(* CODESYS project КАРКАС_СПК_107_М01_07_SP_14_temp-3.project

Project tree, tasks and I/O mapping:
  Device : SPK1xx[M01], Production association OWEN, order no. 4, version 3.5.14.34
    application Application
      libraries: Standard, * (System); ComService, 3.5.4.2 (OWEN); SysCom, 3.5.5.0 (System); ModBus, 3.5.4.3 (Production association OWEN); VisuDialogs, * (System); SysFile, 3.5.9.0 (System); Util, * (System); BASIC, 3.3.3.0 (OSCAT); Visu Utils, 3.5.12.0 (System); AlarmManager, 3.5.14.0 (Intern)
      task VISU_TASK (cyclic, interval 100 ms, priority 30) calls VisuElems.Visu_Prg
      task AlarmManagerTask (cyclic, interval 50 ms, priority 1) calls AlarmManager.Alarm_Prg
      task COM3_TASK (freewheeling, priority 4) calls COM3_PRG
      task MainTask (cyclic, interval t#20ms, priority 5) calls CURRENT_PRG [Обработка непрерывных функций], ASDA_PRG [Обработка алгоритмы работы сервопривода головки]
      task COM2_TASK (freewheeling, priority 3) calls COM2_PRG
      task COM1_TASK (freewheeling, priority 2) calls COM1_PRG [Чтение и запись регистров ASDA-A2 и DVP-SS2]
      program COM3_PRG [ST]
      text list AsdaTextList
      global variables GVL
      STRUCT/
        data type TChiller
        data type TWriteCmd
        data type TSetts
        data type TPulling
        data type TReg
        data type DInt_Word
        data type TModbusRegs
        data type TRWRegs
        data type TAsdaParams
        data type TShnek
        data type TAsda
        data type TReadCmd
        data type TDvp
        data type TPeriod
        data type TPID
        data type TNagrev
        data type TTable
        data type TProject
      SRC_AUX/
        function SWAP_BYTES [ST]
        function BYTES_FROM_DINT [ST]
        function HiWord [ST]
        function LoWord [ST]
        function LoByte [ST]
        function HiByte [ST]
        function BYTES_FROM_INT [ST]
      text list DvpTextList
      SRC_FILE/
        function WRITE_OPTIONS [ST]
        function READ_OPTIONS [ST]
        function RECORD_SAVE [ST]
        function RECS_SELECT [ST]
        function REC_DELETE [ST]
        function REC_EXCHANGE [ST]
        function REC_NAME_EXISTS [ST]
      image pool ImagePool
      SRC/
        program AddReadCmd [ST]
        function SET_FRAME_INDEX_EX [CFC]
        function IsRegValid [ST]
        function ButtonColor [ST]
        program AsdaSetParams [ST]
        function BYTES_FROM_WORD [ST]
        function MERGE_RGB [ST]
        function SET_FRAME_INDEX [CFC]
        program ProcessTempers [ST]
        function WORD_FROM_BYTES [ST]
        function INT_FROM_BYTES [ST]
        function QueuePopReg [ST]
        function QueuePushReg [ST]
        function GET_SET_TEMPERS [ST]
        function block AddWriteCmd_FB [ST]
        function KEYBOARD_STR [ST]
        program ASDA_INIT [ST]
        program ASDA_PARAMS [ST]
        program ASDA_HOMING [ST]
        program ASDA_PULSING [ST]
        program ASDA_SERVO_ON [ST]
        program ASDA_SERVO_OFF [ST]
        program ASDA_PARKING [ST]
        function TERNAR_INT [ST]
        program ASDA_STOP [ST]
        function PENTAR_INT [ST]
        function block PROCESS_DELAY_FB [ST]
      Visu/
        visualisation VIS_SETTS_2
        visualisation Main_Panel
        visualisation DlgConfirm
        visualisation Panel_Reg
        visualisation VIS_MSGS
        visualisation VIS_SETTS_4
        visualisation Setts_Panel
        visualisation VIS_REG
        visualisation VIS_PERIOD
        visualisation VIS_OPERATOR
        visualisation DlgPids
        visualisation VIS_SETTS_1
        visualisation VIS_SETTS_3
        visualisation DlgPulling
        visualisation DlgTargetRegParams
        visualisation DlgConfirmAsdaCMD
        visualisation DlgRegLoad
        visualisation DlgShow
        visualisation DlgKeyboard
        visualisation DlgConfirmSaveAS
        visualisation VIS_EDITOR
        visualisation DlgDeleteRec
      program COM1_PRG [ST]
      global variables GVL_FILE
      program COM2_PRG [ST]
      Alarm Configuration
        alarm class ERR_PCHV (priority 10, acknowledge REP)
        alarm class ERR_PVOZD (priority 10, acknowledge REP)
        text list AG_DVP
        alarm class WARN (priority 10, acknowledge REP)
        alarm group AG_DVP
            1 [ERR_DVP]: Comparison Equal, ExpressionToCompare TRUE, Expression Dvp.E_BITS_si.1 - "Зажим не на исходном концевике"
            2 [ERR_DVP]: Comparison Equal, ExpressionToCompare TRUE, Expression Dvp.E_BITS_si.2 - "Нож не на исходном концевике"
            3 [ERR_DVP]: Comparison Equal, ExpressionToCompare TRUE, Expression Dvp.E_BITS_si.3 - "Превышено время движения зажима"
            4 [ERR_DVP]: Comparison Equal, ExpressionToCompare TRUE, Expression Dvp.E_BITS_si.4 - "Превышено время схода ножа с исходного концевика"
            5 [ERR_DVP]: Comparison Equal, ExpressionToCompare TRUE, Expression Dvp.E_BITS_si.5 - "Превышено время возврата каретки на исходный концевик"
            11 [WARN]: Comparison Equal, ExpressionToCompare FALSE, Expression Dvp.STOP_MANUAL_si - "Нажата аварийная кнопка !"
            7 [ERR_DVP]: Comparison Equal, ExpressionToCompare TRUE, Expression Dvp.E_BITS_si.7 - "РЕЗЕРВ"
            6 [ERR_DVP]: Comparison Equal, ExpressionToCompare TRUE, Expression Dvp.E_BITS_si.6 - "Каретка в крайнем положении"
            8 [WARN]: Comparison Equal, ExpressionToCompare TRUE, Expression Dvp.E_BITS_si.8 - "Превышено время схода каретки с исходного концевика"
            9 [WARN]: Comparison Equal, ExpressionToCompare TRUE, Expression Dvp.E_BITS_si.9 - "Превышено время движения ножа"
            10 [WARN]: Comparison Equal, ExpressionToCompare TRUE, Expression ALARM_MOVE - "Нет движения заготовки в тянущем устройстве"
            0 [ERR_DVP]: Comparison Equal, ExpressionToCompare TRUE, Expression Dvp.E_BITS_si.0 - "Каретка не на исходном концевике"
        text list AG_CONNECT
        alarm group AG_AVAR
            0 [ERR_TEMP]: Comparison Equal, ExpressionToCompare TRUE, Expression Nagrev.E_critical_high - "Превышена критическая температура одной из зон"
            1 [ERR_TEMP]: Comparison Equal, ExpressionToCompare TRUE, Expression Nagrev.E_critical_low - "Температура одной из зон ниже температуры запуска привода"
            2 [WARN]: Comparison Equal, ExpressionToCompare TRUE, Expression Nagrev.E_temp_high - "Превышена температура одной из зон"
            3 [WARN]: Comparison Equal, ExpressionToCompare TRUE, Expression Nagrev.E_temp_low - "Низкая температура одной из зон"
        text list MSGS
        alarm class ERR_CHILLER (priority 10, acknowledge REP)
        alarm class ERR_TEMP (priority 10, acknowledge REP)
        alarm class ERR_DVP (priority 10, acknowledge REP)
        alarm group AG_DEV
            0 [ERR_ASDA]: Comparison Equal, ExpressionToCompare TRUE, Expression Asda.E_CODE.0 - "Сигнал аварии от сервопривода"
            1 [ERR_ASDA]: Comparison Equal, ExpressionToCompare TRUE, Expression Asda.E_CODE.1 - "Сигнал предупреждения от сервопривода"
            2 [ERR_ASDA]: Comparison Equal, ExpressionToCompare TRUE, Expression Asda.E_CODE.2 - "Ошибка инициализации Р2-30 или Р3-06"
            3 [ERR_ASDA]: Comparison Equal, ExpressionToCompare TRUE, Expression Asda.E_CODE.3 - "Превышено время операции HOMING"
            4 [ERR_ASDA]: Comparison Equal, ExpressionToCompare TRUE, Expression Asda.E_CODE.4 - "Превышено время операции ПАРКОВКА"
            5 [WARN]: Comparison Equal, ExpressionToCompare TRUE, Expression Asda.E_CODE.5 - "Ограничение момента сервопривода головки"
            6 [MSG]: Comparison Equal, ExpressionToCompare TRUE, Expression Asda.E_CODE.6 - "Тестовая ошибка"
            7 [ERR_PCHV]: Comparison Equal, ExpressionToCompare TRUE, Expression ALARM_PCHVS.0 - "Аварийный сигнал ПЧВ шнека"
            10 [ERR_PCHV]: Comparison Equal, ExpressionToCompare TRUE, Expression ALARM_PCHVS.8 - "Аварийный сигнал ПЧВ тянущего устройства"
        alarm class MSG (priority 10, acknowledge REP)
        alarm class ERR_ASDA (priority 10, acknowledge REP)
        alarm group AG_CONNECT
            0 [ERR_CONNECT]: Comparison Equal, ExpressionToCompare FALSE, Expression Asda.Connect - "Нет соединение с сервоприводом ASDA-A2"
            1 [ERR_CONNECT]: Comparison Equal, ExpressionToCompare FALSE, Expression Dvp.Connect - "Нет соединения с контроллером DVP"
            2 [ERR_CONNECT]: Comparison Equal, ExpressionToCompare FALSE, Expression Shnek.Connect - "Нет соединения с ПЧВ шнека"
            3 [ERR_CONNECT]: Comparison Equal, ExpressionToCompare FALSE, Expression Pulling.Connect - "Нет соединения с ПЧВ тянущего устройства"
            4 [ERR_CONNECT]: Comparison Equal, ExpressionToCompare FALSE, Expression Chiller.Connect - "Нет соединения с Чиллером"
        text list AG_AVAR
        alarm class ERR_CONNECT (priority 10, acknowledge REP)
        alarm group AG_MSGS
            1 [MSG]: Comparison Equal, ExpressionToCompare TRUE, Expression Dvp.bunker_viveden_msg
            3 [MSG]: Comparison Equal, ExpressionToCompare FALSE, Expression Dvp.Uroven_s_si
            4 [ERR_PVOZD]: Comparison Equal, ExpressionToCompare FALSE, Expression Dvp.PVozd_si
            5 [MSG_PCHV]: Comparison Equal, ExpressionToCompare TRUE, Expression ALARM_PCHVS.1
            11 [MSG_PCHV]: Comparison Equal, ExpressionToCompare TRUE, Expression ALARM_PCHVS.11
            7 [MSG_PCHV]: Comparison Equal, ExpressionToCompare TRUE, Expression ALARM_PCHVS.3
            6 [MSG_PCHV]: Comparison Equal, ExpressionToCompare TRUE, Expression ALARM_PCHVS.2
            12 [MSG_PCHV]: Comparison Equal, ExpressionToCompare TRUE, Expression ALARM_PCHVS.12
            13 [MSG]: Comparison Equal, ExpressionToCompare FALSE, Expression Dvp.Uroven_w_si
            8 [MSG_PCHV]: Comparison Equal, ExpressionToCompare TRUE, Expression ALARM_PCHVS.4
            9 [MSG_PCHV]: Comparison Equal, ExpressionToCompare TRUE, Expression ALARM_PCHVS.9
            10 [MSG_PCHV]: Comparison Equal, ExpressionToCompare TRUE, Expression ALARM_PCHVS.10
            0 [MSG]: Comparison Equal, ExpressionToCompare TRUE, Expression Nagrev.Temper_reached_msg
        text list AG_DEV
        text list AG_CHILLER
        alarm group AG_CHILLER
            11 [ERR_CHILLER]: Comparison Equal, ExpressionToCompare TRUE, Expression Chiller.AlarmFlag1.11 - "Низкая температура нагревания Чиллера"
            21 [ERR_CHILLER]: Comparison Equal, ExpressionToCompare TRUE, Expression Chiller.AlarmFlag2.5 - "Неисправность датчика температуры на выходе Чиллера"
            31 [ERR_CHILLER]: Comparison Equal, ExpressionToCompare TRUE, Expression Chiller.AlarmFlag2.15 - "Обнаружен сигнал контакта входа 2 Чиллера"
            14 [ERR_CHILLER]: Comparison Equal, ExpressionToCompare TRUE, Expression Chiller.AlarmFlag1.14 - "Падение давления на высокой стороне контура хладагента Чиллера"
            24 [ERR_CHILLER]: Comparison Equal, ExpressionToCompare TRUE, Expression Chiller.AlarmFlag2.8 - "Неисправность датчика давления нагнетания Чиллера"
            34 [ERR_CHILLER]: Comparison Equal, ExpressionToCompare TRUE, Expression Chiller.AlarmFlag3.2 - "Неисправен датчик элетрического сопротивления жидкости в Чиллере"
            19 [ERR_CHILLER]: Comparison Equal, ExpressionToCompare TRUE, Expression Chiller.AlarmFlag2.3 - "Ошибка памяти контроллера Чиллера"
            29 [ERR_CHILLER]: Comparison Equal, ExpressionToCompare TRUE, Expression Chiller.AlarmFlag2.13 - "Обслуживание компрессора двигателя Чиллера"
            17 [ERR_CHILLER]: Comparison Equal, ExpressionToCompare TRUE, Expression Chiller.AlarmFlag2.1 - "Перегрузка компрессора Чиллера"
            27 [ERR_CHILLER]: Comparison Equal, ExpressionToCompare TRUE, Expression Chiller.AlarmFlag2.11 - "Обслуживание насоса Чиллера"
            12 [ERR_CHILLER]: Comparison Equal, ExpressionToCompare TRUE, Expression Chiller.AlarmFlag1.12 - "Высокое давление нагнетания компрессора Чиллера"
            22 [ERR_CHILLER]: Comparison Equal, ExpressionToCompare TRUE, Expression Chiller.AlarmFlag2.6 - "Неисправность датчика температуры на входе Чиллера"
            32 [ERR_CHILLER]: Comparison Equal, ExpressionToCompare TRUE, Expression Chiller.AlarmFlag3.0 - "Обнаружена утечка воды Чиллера"
            15 [ERR_CHILLER]: Comparison Equal, ExpressionToCompare TRUE, Expression Chiller.AlarmFlag1.15 - "Повышение давления на низкой стороне контура хладагента Чиллера"
            25 [ERR_CHILLER]: Comparison Equal, ExpressionToCompare TRUE, Expression Chiller.AlarmFlag2.9 - "Неисправность датчика давления нагнетания компрессора Чиллера"
            16 [ERR_CHILLER]: Comparison Equal, ExpressionToCompare TRUE, Expression Chiller.AlarmFlag2.0 - "Падение давления на низкой стороне контура хладагента Чиллера"
            10 [ERR_CHILLER]: Comparison Equal, ExpressionToCompare TRUE, Expression Chiller.AlarmFlag1.10 - "Низкая температура на входе компрессора Чиллера"
            20 [ERR_CHILLER]: Comparison Equal, ExpressionToCompare TRUE, Expression Chiller.AlarmFlag2.4 - "Сработал предохранитель постоянного тока в Чиллере"
            30 [ERR_CHILLER]: Comparison Equal, ExpressionToCompare TRUE, Expression Chiller.AlarmFlag2.14 - "Обнаружен сигнал контакта входа 1 Чиллера"
            13 [ERR_CHILLER]: Comparison Equal, ExpressionToCompare TRUE, Expression Chiller.AlarmFlag1.13 - "Unused"
            23 [ERR_CHILLER]: Comparison Equal, ExpressionToCompare TRUE, Expression Chiller.AlarmFlag2.7 - "Неисправность датчика температуры на входе компрессора Чиллера"
            33 [ERR_CHILLER]: Comparison Equal, ExpressionToCompare TRUE, Expression Chiller.AlarmFlag3.1 - "Повышение элетрического удельного сопротивления жидкости в Чиллере"
            18 [ERR_CHILLER]: Comparison Equal, ExpressionToCompare TRUE, Expression Chiller.AlarmFlag2.2 - "Ошибка связи с контроллером Чиллера"
            28 [ERR_CHILLER]: Comparison Equal, ExpressionToCompare TRUE, Expression Chiller.AlarmFlag2.12 - "Обслуживание вентилятора двигателя Чиллера"
            8 [ERR_CHILLER]: Comparison Equal, ExpressionToCompare TRUE, Expression Chiller.AlarmFlag1.8 - "Падение давления нагнетания Чиллера"
            9 [ERR_CHILLER]: Comparison Equal, ExpressionToCompare TRUE, Expression Chiller.AlarmFlag1.9 - "Высокая температура на входе компрессора Чиллера"
            26 [ERR_CHILLER]: Comparison Equal, ExpressionToCompare TRUE, Expression Chiller.AlarmFlag2.10 - "Неисправность датчика давления на входе компрессора Чиллера"
            0 [ERR_CHILLER]: Comparison Equal, ExpressionToCompare TRUE, Expression Chiller.AlarmFlag1.0 - "Низкий уровень воды в Чиллере"
            1 [ERR_CHILLER]: Comparison Equal, ExpressionToCompare TRUE, Expression Chiller.AlarmFlag1.1 - "Высокая температура воды на выходе Чиллера"
            2 [ERR_CHILLER]: Comparison Equal, ExpressionToCompare TRUE, Expression Chiller.AlarmFlag1.2 - "Температура на выходе Чиллера выросла"
            3 [ERR_CHILLER]: Comparison Equal, ExpressionToCompare TRUE, Expression Chiller.AlarmFlag1.3 - "Температура на выходе Чиллера..."
            4 [ERR_CHILLER]: Comparison Equal, ExpressionToCompare TRUE, Expression Chiller.AlarmFlag1.4 - "Высокая температура воды на входе Чиллера"
            5 [ERR_CHILLER]: Comparison Equal, ExpressionToCompare TRUE, Expression Chiller.AlarmFlag1.5 - "Высокая давление нагнетания Чиллера"
            6 [ERR_CHILLER]: Comparison Equal, ExpressionToCompare TRUE, Expression Chiller.AlarmFlag1.6 - "Ненормальная работа насоса Чиллера"
            7 [ERR_CHILLER]: Comparison Equal, ExpressionToCompare TRUE, Expression Chiller.AlarmFlag1.7 - "Повышение давления нагнетания Чиллера"
        alarm class MSG_PCHV (priority 10, acknowledge REP)
        text list AlarmGroup
        alarm group AlarmGroup
      program CURRENT_PRG [ST]
      text list FileTextList
      program ASDA_PRG [ST]
    Network : Network, Production association OWEN, version 3.5.14.3001
        unmapped channels: DHCP enabled, IP, Mask, Gateway, MAC, Hostname, Enable DHCP, New IP, New Mask, New Gateway, New Hostname, Set Settings
    Drives : Drives, Production association OWEN, version 3.5.14.3001
        input  Application.MMCMounted : BIT  // MMC Mounted
        output Application.EnableDrivers : BIT  // Enable Drives
        output Application.bUnmount : BIT  // MMC Unmount
        unmapped channels: FS size, FS used, FS free, USB Mounted, USB Unmount done, USB size, USB used, USB free, MMC Unmount done, MMC size, MMC used, MMC free, USB Unmount
    Buzzer : Buzzer, Production association OWEN, version 3.5.14.3001
        unmapped channels: Buzzer enabled, Enable Buzzer
    Info : Info, Production association OWEN, version 3.5.14.3001
        input  Application.Project.sVendor : ARRAY [0..80] OF BYTE  // VENDOR
        input  Application.Project.sName : ARRAY [0..80] OF BYTE  // DEVICE
        input  Application.Project.sSerial : ARRAY [0..80] OF BYTE  // SERIAL
        input  Application.Project.sRuntime : ARRAY [0..80] OF BYTE  // RUNTIME
        input  Application.Project.sFirmwareVersion : ARRAY [0..80] OF BYTE  // FIRMWARE
        input  Application.Project.sLinuxVersion : ARRAY [0..80] OF BYTE  // LINUX
        input  Application.Project.sNeedTarget : ARRAY [0..80] OF BYTE  // TARGET
        unmapped channels: PROJECT, AUTHOR, VERSION, PROFILE, LASTCHANGES
    Debug : Debug, Production association OWEN, version 3.5.14.3001
        unmapped channels: RAM used, RAM free, Open files, Processor usage, Core temp, Enable Debug, Debug pause
    OwenCloud : OwenCloud, Production association OWEN, version 3.5.14.3002
        unmapped channels: OwenCloud enabled, Folder error, Symbol error, No Symbol Config, Status, Enable OwenCloud
    Screen : Screen, Production association OWEN, version 3.5.14.3001
        unmapped channels: Get Brightness, Dim time, Off time, Full brightness, Dim brightness, Off brightness, Dim visu name, Off visu name, On visu name, Wake up
    OwenRTC : OwenRTC, Production association OWEN, version 3.5.14.3001
        unmapped channels: Year, Month, Day, Hour, Minute, Second, Day of Week, Week of Year, Format Date, Format Time, UTC Offset, NTP Enabled, NTP Error, System Timer, Date And Time, New Year, New Month, New Day, New Hour, New Minute, New Second, New UTC Offset, Set Settings DT, Enable NTP, Prefer Server
    Watchdog : Watchdog, Production association OWEN, version 3.5.14.3001
        unmapped channels: Exception Handling, Last Exception Code, Last Exception Description, Last Exception Time, Hardware Watchdog Flag, Power Reboot Count, Watchdog Reboot Count, Exception Reboot Count, Command Reboot Count, Reboot, Reset Counters
  5ce3da45-db07-42e7-a21c-a00fff4ed8f6|Images\Banned.png
  5ce3da45-db07-42e7-a21c-a00fff4ed8f6|Images\crosscirclehd.png
  5ce3da45-db07-42e7-a21c-a00fff4ed8f6|Images\Good.png
  5ce3da45-db07-42e7-a21c-a00fff4ed8f6|Images\Dialog_win_7_800x480.jpg
  5ce3da45-db07-42e7-a21c-a00fff4ed8f6|Images\Dialog_win_7_400x200.jpg
  5ce3da45-db07-42e7-a21c-a00fff4ed8f6|Images\iError.png
  5ce3da45-db07-42e7-a21c-a00fff4ed8f6|Images\tickcirclehd.png
  5ce3da45-db07-42e7-a21c-a00fff4ed8f6|Images\danger.png
  5ce3da45-db07-42e7-a21c-a00fff4ed8f6|Images\Dialog_win_7_600x300.jpg
  text list GlobalTextList
  5ce3da45-db07-42e7-a21c-a00fff4ed8f6|Images\Warning.png
  5ce3da45-db07-42e7-a21c-a00fff4ed8f6|Images\Dialog_win_7_700x380.jpg
  5ce3da45-db07-42e7-a21c-a00fff4ed8f6|Images\Dialog_win_7_750x450.jpg
*)

// Device/Application/STRUCT/TChiller
TYPE TChiller :
STRUCT
	Connect			: BOOL;			// Флаг соединения с Чиллером
	T_ACTUAL		: REAL;
	
	Pusk			: BOOL;
	Block			: BOOL;
	AVAR			: BOOL;			// Флаг аварии Чиллера (читаем по RS-485)
	Status			: WORD;
	Status_2		: WORD;

	AlarmFlag1		: WORD;			// Флаги аварии Чиллера
	AlarmFlag2		: WORD;
	AlarmFlag3		: WORD;

	FillColor		: DWORD;		(* Цвет заливки окошка температуры *)
	FrameColor		: DWORD;		(* Цвет контура окошка температуры *)

	BtnFillColor	: DWORD;		(* Цвет заливки площадок кнопок ПУСК в автоматическом режиме *)
	BtnFrameColor	: DWORD;		(* Цвет контура площадок кнопок ПУСК в автоматическом режиме *)
	
END_STRUCT
END_TYPE

(*
Status flag

0	Run flag						Run status (Include the independent operation of the pump) 0= Stop 1= Run
1	Operation stop alarm flag		Operation stop alarm given off status 0= Not occurred 1= Operation stop alarm given off
2 	Operation continued alarm flag	Operation continued alarm given off status 0= Not occurred 1= Operation continued alarm given off
3	Unused
4	Press Unit flag					Pressure unit set status 0= MPa 1= PSI
5	Remote status flag				Remote status 0= Other than SERIAL mode 1= SERIAL mode
6	Unused
7	Unused
8	Unused
9	Completion of preparation		Completion of preparation (TEMP READY) status
	(TEMP READY) flag				0= Condition isn’t formed 1= Condition is formed
10	Temperature unit flag			Temperature unit set status 0= Centigrade (oC) 1= Fahrenheit (oF)
11	Run timer flag					Run timer set status 0= Not set 1= Set
12	Stop timer flag					Stop timer set status 0= Not set 1= Set
13	Reset after power failure flag	Reset after power failure set status 0= Not set 1= Set
14	Anti-freezing flag				Anti-freezing set status 0= Not set 1= Set
15	Automatic fluid filling flag	Automatic fluid filling condition 0= Stop 1= Fluid ∗ The signal of the product without an option [Automatic filling] also changes.

Status flag 2
0-1	Electric resistivity/			Electric resistivity/conductivity setting status conductivity setting flag
									0= Not set 1= Electric resistivity is set 2= Electric conductivity is set
2-15	Unused
*)

// Device/Application/STRUCT/TWriteCmd
TYPE TWriteCmd :
(
	wcAsda_P2_30:=0,
	wcAsda_P3_06,
	wcAsda_P4_07_1,
	wcAsda_P4_07_2,
	wcAsda_P4_07_3,
	wcAsda_P4_07_4,
	
	wcAsdaParams,
	wcAsda_Homing,
	wcAsda_Forward,
	wcAsda_Backward,
	wcAsda_Parking,
	wcAsda_Working,
	wcAsda_Stop,
	
	wcChiller_Ust,
	wcChiller_Start,
	wcChiller_Stop,
	
	wcShnek_Ust,
	wcShnek_Start,
	wcShnek_Stop,
	
	wcPulling_Ust,
	wcPulling_Start,
	wcPulling_Stop
);
END_TYPE

// Device/Application/STRUCT/TSetts
TYPE TSetts :
STRUCT
	T_ZAP					: ARRAY [0..NUM_TEMPS-1] OF REAL;		// Температуры запуска приводов
	TM_VIGON				: WORD;		// Время выгона массы в секундах	
	otkl_alarm_zvuk			: BOOL;		// Флаг отключения звуковой сигнализации аварий
	otkl_h_temp				: BOOL;		// Переменная для отключения ошибки "Превышение температуры одной из зон"
	otkl_l_temp				: BOOL; 	// Переменная для отключения ошибки "Низкая температура одной из зон" 
	otkl_c_pulling			: BOOL;		// Переменная для отключения контроля движения ТЯУ
	use_vigon				: BOOL;		// Флаг выгона массы
	use_bunker				: BOOL;		// Флаг использования бункера
	use_servo_without_temp	: BOOL;		// Разрешить работу головки без разогрева (ТОЛЬКО ДЛЯ ОТЛАДКИ !!!)
	use_shnek_without_temp	: BOOL;		// Разрешить работу шнека без разогрева (ТОЛЬКО ДЛЯ ОТЛАДКИ !!!)
	
	CondEnableZones1_4		: BOOL;		// Флаг для условного включения зон 1-4
	CondIZone				: BYTE;		// Номер зоны (5-7), по которой управляется включение зон 1-4
	CondValue				: REAL;		// Значение 0-100 % от температуры уставки зоны (5-7), при превышении которой включаются зоны 1-4

	REP_MM					: REAL;		// Начальное положение (смещение) реперной точки относительно заднего концевика в 0.01 мм
	TimeVigon				: WORD;		// Время выгона массы после вывода бункера в секундах
	K_Length				: REAL;		// Длина заготовки в мм
	zd_temps				: ARRAY [0..NUM_TEMPS-1] OF REAL;	// Температуры для автонастройки ПИД-регуляторов

END_STRUCT
END_TYPE

// Device/Application/STRUCT/TPulling
TYPE TPulling :
STRUCT
	Connect			: BOOL;			(* Флаг соединения *)
	Pusk			: BOOL;			(* Флаг включения *) 
	Block			: BOOL;			(* Блокировка тянущего *)
	STW				: WORD;			(* Слово состояния *)
	MAV				: WORD;			(* Основное текущее значение привода *)
	
	Speed			: REAL;			(* Реальная скорость движения в процентах *)
	ActiveParamSet	: WORD;			(* Активный набор данных в ПЧВ *)
	BtnFillColor	: DWORD;		(* Цвет заливки площадок кнопок ПУСК в автоматическом режиме *)
	BtnFrameColor	: DWORD;		(* Цвет контура площадок кнопок ПУСК в автоматическом режиме *)
	
	
END_STRUCT
END_TYPE

(* ПЧВ ТЯУ использует 2 набора параметров:
Набор параметров 1 - для работы без обратной связи,
Набор параметров 2 - для работы с обратной связью и ПИ-регулятором *)

(*
1. Обороты двигателя ТЯУ при 50 Гц = 1350 об/мин
2. Редуктор - к-т редукции = 304
3. Обороты вала редуктора = 1350/304 = 4,44 об/мин
4. Число зубов ведущей шестерёнки = 11
5. Число зубов ведомой шестерёнки = 20
6. Обороты вала ведомой шестерёнки (тянущего вала) = 4,44*(11/20) = 2,4424 об/мин
7. Диаметр тянущего вала = 97 мм
8. Диаметр шкива энкодера = 63,6 мм
9. Обороты вала энкодера = 2,4424*(97/63,6) = 3,725 об/мин
10. Обороты энкодера в секунду = 3,725,60 = 0,06208 об/сек
11. Частота импульсов энкодера = 0,06208*5000 = 310,425 Гц
12. МАКСИМАЛЬНАЯ ЧАСТОТА ЭНКОДЕРА (при питающей частоте двигателя 100 Гц) = 310,425*100/50 = 620,849 Гц

*)

// Device/Application/STRUCT/TReg
TYPE TReg :
STRUCT
	Name		: STRING (64);						// Имя режима
	Desc		: STRING (64);						// Примечание

	TEMPS		: ARRAY [0..NUM_TEMPS-1] OF REAL;	// Уставки температур зон нагрева 0-6
	T_MASS		: REAL;								// Температура массы
	T_CHIL		: REAL;								// Уставка температуры Чиллера
	Period		: TPeriod;							// Параметры периода работы головки
	
	Qm			: REAL;		// Производительность шнека в процентах (возможно далее в г/мин после экспериментального создания шкалы)
	Speed		: REAL;		// Скорость движения тянущего устройства в процентах (возможно далее в мм / сек)
	Freq		: REAL;		// Частота колебаний коронки, Гц 
	
	REZ_1		: REAL;		// Резерв 1
	REZ_2		: REAL;		// Резерв 2
	REZ_3		: REAL;		// Резерв 3
	
END_STRUCT
END_TYPE

// Device/Application/STRUCT/DInt_Word
TYPE DInt_Word :
UNION

	dDInt	: DINT;
	wWord	: ARRAY[0..1] OF WORD;
	
END_UNION
END_TYPE

// Device/Application/STRUCT/TModbusRegs
TYPE TModbusRegs :
STRUCT
	DevAdr		: BYTE;						// Адрес устройства
	RegAdr		: WORD;						// Адрес регистра
	pVals		: POINTER TO WORD;			// Указатели на переменные (для чтения и записи)
	RegsCount	: BYTE;						// Число регистров записи или чтения
END_STRUCT
END_TYPE

// Device/Application/STRUCT/TRWRegs
TYPE TRWRegs :
STRUCT
	REGS	: ARRAY [0..MAX_MODBUS_REGS-1] OF TModbusRegs;		// Структура для последовательной записи
	Count	: BYTE;												// Счётчик для обработки цикла

END_STRUCT
END_TYPE

// Device/Application/STRUCT/TAsdaParams
//{attribute 'qualified_only'}
//{attribute 'strict'}
TYPE TAsdaParams :
(
	ap_Accs,
	ap_Speeds,
	ap_Dels,
	ap_Dists
);
END_TYPE

// Device/Application/STRUCT/TShnek
TYPE TShnek :
STRUCT
	Connect		: BOOL;			(* Флаг соединения *)
	Pusk		: BOOL;			(* Флаг включения *) 
	Block		: BOOL;			(* Блокировка шнека *)
	STW			: WORD;			(* Слово состояния *)
	MAV			: WORD;			(* Основное текущее значение привода *)
	
	Qm			: REAL;			(* Реальная производительность в процентах *)
	
	FillColor	: DWORD;		(* Цвет заливки площадок кнопок ПУСК в автоматическом режиме *)
	FrameColor	: DWORD;		(* Цвет контура площадок кнопок ПУСК в автоматическом режиме *)

END_STRUCT
END_TYPE

(* Слово состояния STW
---------------------------------------------------------------------
		|		1										|		0
----------------------------------------------------------------------
STW.0	|	Готовность к управлению					|	Управление не готово
STW.1	|	Привод готов							|	Привод не готов
STW.2	|	Нет останова выбегом					|	Останов выбегом
STW.3	|	Аварийный сигнал						|	Нет аварийного сигнала
STW.4	|	Есть отображение ошибки на ЛПО			|	Нет отображения ошибки на ЛПО
STW.5	|	НЕ ИСПОЛЬЗУЕТСЯ							|
STW.6	|	Отключение с блокировкой				|	Нет критических аварий
STW.7	|	Предупреждение							|	Нет предупреждения
STW.8	|	На задании								|	Не на задании (например, разгон)
STW.9	|	Автоматический режим					|	Ручной режим
STW.10	|	В частотном диапазоне					|	Вне частотного диапазона
STW.11	|	Работа									|	Остановлен
STW.12	|	Останов с автоматическим перезапуском	|	Привод в норме
STW.13	|	Предупреждение о напряжении				|	Нет предупреждения о напряжении
STW.14	|	Предел по току							|	Нет предела по току
STW.15	|	Предупреждение о перегреве				|	Нет предупреждения о перегреве

*)

// Device/Application/STRUCT/TAsda
TYPE TAsda :
STRUCT
	Connect			: BOOL;			// Флаг соединения с ASDA-A2
	IsInit			: BOOL;			// Флаг
	IsHoming		: BOOL;			// Флаг нахождения реперной точки
	IsServo_ON		: BOOL;			// Фгаг включенного сервопривода
	DoPulsing		: BOOL;			// Флаг процесса пульсирования
	AllowManual		: BOOL;			// Флаг разрешения ручного режима
	P0_01			: WORD;			// Код ошибки (для логического дополнения до 6 читаемых регистров одной командой через Mapping)
	P0_46			: WORD;			// Параметр P0-46 - состояние дискретных выходов
	P2_30			: WORD;			// Параметр Р2-30 - отключение EEPROM (д.б=5)
	P3_06			: WORD;			// Параметр Р3-06 - способ управления дискретными входами (д.б.=3)
	P4_07			: WORD;			// Параметр Р4-07 - состояние дискретных входов
	P5_07			: WORD;			// Параметр Р5-07 - управление PR - циклическое чтение
	E_CODE			: WORD:=0;		// Код ошибки сервопривода
	WAIT			: BOOL;			// Флаг состояния ожидания
	WAIT_ERR		: BOOL;			// Флаг ожидания команды сброса аварии
	WAIT_WORK		: BOOL;			// Флаг нахождения в состоянии работы
	Pusk			: BOOL;			// Флаг работы в пульсирующем режиме
	Block			: BOOL;			// Блокировка головки
	Torque			: INT;			// Текущий момент
	TorqueMin		: INT;			// Минимальный момент
	TorqueMax		: INT;			// Максимальный момент
	
	// Вспомогательные переменные
	BtnFillColor	: DWORD;	(* Цвет заливки площадок кнопок ПУСК в автоматическом режиме *)
	BtnFrameColor	: DWORD;	(* Цвет контура площадок кнопок ПУСК в автоматическом режиме *)

	text_id			: BYTE;			// Индекс сообщения в списке сообщений - 
	E_ALARM			: WORD;			// Код ошибки сервопривода после перевода из BCD
	
END_STRUCT
END_TYPE

(* Состояние дискретных входов
P4-07.0		- Servo ON
P4-07.1		- Alarm Reset
P4-07.2		- Reverse LIM
P4-07.3		- Forward LIM
*)

(* Коды ошибок сервопривода
E_CODE.0	- SP - сигнал ALRM
E_CODE.1	- SP - сигнал WARN
E_CODE.2	- SP - Ошибка инициализации Р2-30 или Р3-06
E_CODE.3	- SP - Превышено время операции HOMING
E_CODE.4	- SP - Превышено время операции PARKING
E_CODE.5	- SP - Превышение момента
E_CODE.6	- SP - Тестовая ошибка
*)
(* Значения P0-46 (дискретные выходы)
SP_P0_46.0	- SRDY (Готовность привода)
SP_P0_46.1	- SON (Servo On - привод работает)
SP_P0_46.2	- ZSPD (Нулевая скорость)
SP_P0_46.3	- TSPD (Скорость достигнута)
SP_P0_46.4	- TPOS (Зад. положение достигнуто)
SP_P0_46.5	- TQL (Ограничение момента)
SP_P0_46.6	- ALRM (Авария привода)
SP_P0_46.7	- BRKR (Управление тормозом)
SP_P0_46.8	- HOME (Исходное положение достигнуто)
SP_P0_46.9	- OLW (Предупреждение о перегрузке)
SP_P0_46.10	- WARN (Предупреждение активно. WARN активизируется, во время ограничения прямого или обратного вращения;
аварийного стопа, ошибки коммуникации, и при низком напряжении питания.)*)

// Device/Application/STRUCT/TReadCmd
//{attribute 'qualified_only'}
//{attribute 'strict'}
TYPE TReadCmd :
(
	rcAsda_P2_30:=0,		// Дополнительные функции входов		
	rcAsda_P3_06,			// Функция управления входными сигналами
	rcAsda_P6_01			// Положение реперной точки относительно заднего концевика
	
);
END_TYPE

// Device/Application/STRUCT/TDvp
TYPE TDvp :
STRUCT
	Connect				: BOOL;		// Флаг соединения
	bunker_viveden_msg	: BOOL;		// Оповещатель "Бунер выведен !!!"

	Nasos_so			: BOOL;		// Сигнал включения насоса
	Nasos_OTL			: BOOL;		// Флаг отладочного включения насоса

	Uroven_s_si			: BOOL;		// Уровень сырья в бункере
	Uroven_w_si			: BOOL;		// Уровень воды в баке

	Bunker_si			: BOOL;		// Положение бункера
	PVozd_si			: BOOL;		// Давление воздуха
	KarIsx_si			: BOOL;		// Датчик исходного положения каркаса
	KarRab_si			: BOOL;		// Датчик рабочего положения каркаса
	ZazhIsx_si			: BOOL;		// Датчик исходного положения зажима
	KnifeIsx_si			: BOOL;		// Датчик исходного положения ножа
	KnifeRab_si			: BOOL;		// Датчик рабочего положения ножа

	Nasos_si			: BOOL;		// Реле включения насоса
	Karet_si			: BOOL;		// Пневмоцилиндр каретки
	Zazh_si				: BOOL;		// Пневмоцилиндр зажима
	Knife_si			: BOOL;		// Пневмоцидиндр ножа
	F_OTR_si			: BOOL;		// Импульс отрезки заготовки
	STOP_MANUAL_si		: BOOL;		// Сигнал аварийного останова от кнопки СТОП (ИНВЕРСНЫЙ)
	E_BITS_si			: WORD;		// Биты ошибок от DVP

	Pids				: ARRAY [0..NUM_TEMPS-1] OF TPID;		// Параметры ПИД-регуляторов
	pid_index			: WORD;		// Переменная для выбора индекса 0-6 ПИД-регулятора
	zone_index			: WORD;		// Переменная для выбора номера зоны 1-7 ПИД-регулятора
	pid_read			: BOOL;		// Переменная импульса чтения ПИД
	pid_write			: BOOL;		// Переменная импульса записи ПИД
	
	zd_selector			: BOOL;		// Переключатель - откуда брать задания температур для настройки ПИД
	AutoPIDActivate		: BOOL;		// Переменная для активизации автонастройки ПИД
	
	Encoder				: BOOL;		// Флаг вращения энкодера
END_STRUCT
END_TYPE

// Device/Application/STRUCT/TPeriod
TYPE TPeriod :
STRUCT
	Per_FirstHP		: REAL;						// Процент первого полупериода (второй - остаток)
	Per_Pulses		: ARRAY [0..1] OF REAL;		// Проценты импульсов 1-го и 2-го полупериодов в соотв. полупериодах	
	Per_Levels		: ARRAY [0..1] OF REAL;		// Проценты уровней 1-го и 2-го полупериодов в соотв. импульсах
	Offsets			: ARRAY [0..1] OF REAL;		// милиметры, P6-21 - Смещение вперёд, P6-23 - назад от реперной точки
	
END_STRUCT
END_TYPE

(* Единицы измерения
Accs		- милисекунды
Speeds		- обороты в минуту
Dels		- милисекунды
Offsets		- PUU
*)

// Device/Application/STRUCT/TPID
TYPE TPID :
STRUCT
	formula		: WORD;			// Формула ПИД-регулятора (0-независимая, 1-зависимая см. документацию на температурный модуль)
	Kc_Kp		: REAL;			// Пропорциональный коэффициент
	Ti_Ki		: REAL;			// Коэффициент интегрирования
	Td_Kd		: REAL;			// Коэффициент дифференцирования
	Tf			: REAL;			// Постоянная времени дифференцирования
	
END_STRUCT
END_TYPE

// Device/Application/STRUCT/TNagrev
TYPE TNagrev :
STRUCT
	T_Actuals			: ARRAY [0..NUM_TEMPS-1] OF REAL;	// Текущие температуры
	T_ActualMass		: REAL;			// Текущая температура массы
	T_Enables_si		: WORD;			// Биты включенных зон (из Dvp (не используются))
	T_Enables			: WORD;			// Биты заданных включенных зон

	Auto_IN				: BYTE;			// Вспомогательная переменные для сборки сигналов автонастройки от Dvp 
	Auto_OUT			: BYTE;			// Вспомогательная переменная для сборки сигналов автонастройки к Dvp

	E_critical_high		: BOOL;			// Флаг критической температуры одной из зон
	E_critical_low		: BOOL;			// Флаг температуры одной из зон ниже температуры запуска приводов
	E_temp_high			: BOOL;			// Флаг превышения температуры одной из зон
	E_temp_low			: BOOL;			// Флаг низкой температуры одной из зон
	Temper_Reached		: BOOL;			// Флаг выхода на темрературный режим
	Temper_Reached_msg	: BOOL;			// Оповещатель достижения температуры
	Nagrev_on			: BOOL;			// Флаг включения нагревателей
	NagrevFillColor		: DWORD;		// Цвет заливки площадок кнопок ПУСК в автоматическом режиме
	NagrevFrameColor	: DWORD;		// Цвет контура площадок кнопок ПУСК в автоматическом режиме
	FillColors			: ARRAY [0..NUM_TEMPS-1] OF DWORD;	// Массив цветов заливок
	FrameColors			: ARRAY [0..NUM_TEMPS-1] OF DWORD;	// Массив цветов фреймов
	FillColorMass		: DWORD;		// Цвет заливки окошка температуры массы
	FrameColorMass		: DWORD;		// Цвет контура окошка температуры массы

	text_id				: BYTE;			// Индекс текста из списка состояний

END_STRUCT
END_TYPE

// Device/Application/STRUCT/TTable
TYPE TTable :
STRUCT
	Recs		: ARRAY [0..TABLE_NUM_ROWS-1] OF TReg;	// Записи таблицы
	RowCount	: INT;	// Число строк таблицы, RowCount-1 - максимальный индекс массива для таблицы
	RowSel		: INT;	// Выделеная строка в таблице
	PageNum		: INT;	// Номер страницы в таблице 
	NumFileRecs	: INT;	// Суммарное число записей в таблице
	iMsg		: BYTE;	// Флаг сообщений при загрузке таблицы

END_STRUCT
END_TYPE

// Device/Application/STRUCT/TProject
TYPE TProject :
STRUCT
	sVendor				: STRING;	// Производитель
	sName				: STRING;	// Имя
	sSerial				: STRING;	// Серийный номер	
	sRuntime			: STRING;	// Рабочая версия
	sFirmwareVersion	: STRING;	// Информация о прошивке
	sNeedTarget			: STRING;	// Требуемый таргет-файл
	sLinuxVersion		: STRING;	// Версия ОС Linux в контроллере
	
	
	
END_STRUCT
END_TYPE

// Device/Application/GVL
VAR_GLOBAL CONSTANT

ADR_DVP			: BYTE:=1;		// Modbus адрес контроллера DVP на линии COM_1 
ADR_ASDA		: BYTE:=64;		// Modbus адрес сервопривода ASDA на линии COM_1
ADR_SHNEK		: BYTE:=24;		// Modbus адрес  частотника шнека на линии COM_2
ADR_PULLING		: BYTE:=32;		// Modbus адрес  частотника тянущего устройства на линии COM_2
ADR_CHILLER		: BYTE:=80;		// Modbus адрес  Чиллера на линии COM_3

FREQ_MIN		: REAL:=0.1;	// Минимальная частота головки
FREQ_MAX		: REAL:=5.0;	// Максимальная частота головки

NUM_TEMPS 		: BYTE:=7;		// Размер массива температур зон нагрева
T_CRITICALS		: ARRAY [0..NUM_TEMPS-1] OF REAL:=[280,380,380,380,380,380,380];		// Критические температуры зон 1,2,3,4,5,6,7 соответственно
T_CHIL_CRITICAL	: REAL:=50;																// Критическая температура Чиллера

T_MAXS_ZAD		: ARRAY [0..NUM_TEMPS-1] OF REAL:=[250,350,350,350,350,350,350];		// Максимальные температуры задания зон 1,2,3,4,5,6,7 соответственно
T_MINS_ZAD		: ARRAY [0..NUM_TEMPS-1] OF REAL:=[100,100,100,100,100,100,100];		// Минимальные температуры задания зон 1,2,3,4,5,6,7 соответственно

T_ZAP_MIN		: REAL:=200;			// !!!!!!!!!!!!!!!!!!!!!!
T_ZAP_MAX		: REAL:=300;

T_MAX_MASS_ZAD	: REAL:=350;	// Максимальная температура задания для массы
T_MIN_MASS_ZAD	: REAL:=200;	// Минимальная температура задания для массы

T_MAX_CHIL_ZAD	: REAL:=40;		// Максимальная температура задания для Чиллера
T_MIN_CHIL_ZAD	: REAL:=8;		// Минимальная температура задания для Чиллера

DT_MINS			: ARRAY [0..NUM_TEMPS-1] OF REAL:=[3,3,3,3,3,3,3];	// +- 3 градуса от номинала считаем норма
DT_MASS_MIN		: REAL:=3;
DT_CHIL_MIN		: REAL:=2;

DT_MAXS			: ARRAY [0..NUM_TEMPS-1] OF REAL:=[7,7,7,7,7,7,7];	// +- 7 за границей DT_MAX ошибка (красная), между DT_MAX и DT_MIN предупреждение(оранжевая), до DT_MIN - норма(зелёная)
DT_MASS_MAX		: REAL:=7;
DT_CHIL_MAX		: REAL:=5;

ASDA_HP_MIN		: REAL:=10;		// Минимальное значение "полупериода" в процентах от периода частоты колебаний коронки		
ASDA_HP_MAX		: REAL:=90;		// Максимальное значение "полупериода" в процентах от периода частоты колебаний коронки

ASDA_PULSE_MIN	: REAL:=20;		// Минимальное значение импульса в процентах от "полупериода"
ASDA_PULSE_MAX	: REAL:=100;	// Максимальнон значение импульса в процентах от "полупериода"

ASDA_LEVEL_MIN	: REAL:=20;		// Минимальный уровент внутри импульса "полупериода"
ASDA_LEVEL_MAX	: REAL:=80;		// Максимальный уровент внутри импульса "полупериода"

LEN_MIN			: REAL:=200;	// Минимальная длина каркаса в мм
LEN_MAX			: REAL:=3000;	// Максимальная длина каркаса в мм

SPEED_MIN		: REAL:=0.0;	// Минимальное значение скорости в процентах
SPEED_MAX		: REAL:=100.0;	// Максимальное значение скорости в процентах

QM_MIN			: REAL:=0.0;	// Минимальное значение производительности в процентах
QM_MAX			: REAL:=100.0;	// Максимальное значение производительности в процентах

PUU_PER_MM		: REAL:=20000;	// 20 0000 - Число PUU на перемещение 1 мм
REP_MIN			: REAL:=-9.5;	// Минимальное положение реперной точки относительно заднего концевика в 0.01 мм
REP_MAX			: REAL:=1.0;	// Максимальное положение реперной точки относительно заднего концевика в 0.01 мм
WORK_SIZE		: REAL:=12;		// Максимальный рабочий ход

MAX_MODBUS_REGS	: WORD:=128;

REG_DEF			: TReg:=
(
	Name:='default',		// Имя режима
	Desc:='description',	// Примечание

	TEMPS:=[
		185,	(* PID1, температура 1 зоны *)
		225,	(* PID2, температура 2 зоны *)
		240,	(* PID3, температура 3 зоны *)
		245,	(* PID4, температура 4 зоны *)
		225,	(* PID5, температура 5 зоны *)
		245,	(* PID6, температура 6 зоны *)
		240		(* PID7, температура 7 зоны *)
	],
	
	T_MASS:=230,						// Температура массы
	
	T_CHIL:=20,							// Температура Чиллера

	Period:= (
		Per_FirstHP		:= 50,			// Процент первого полупериода (второй - остаток)
		Per_Pulses		:= [50,50],		// Проценты импульсов в соответствующих полупериодах
		Per_Levels		:= [75,75],		// Проценты уровней внутри импульсов		
		Offsets			:= [-0.5, -3.0]	// мм
	),

	Qm					:= 62,			// Производительность шнека в процентах (возможно далее в г/мин после экспериментального создания шкалы)
	Speed				:= 36.5,		// Скорость движения заготовки в процентах (возможно далкк в мм / сек)
	Freq				:= 1.82,			// Герц

	REZ_1				:= 0,			// РЕЗЕРВ 1
	REZ_2				:= 0,			// РЕЗЕРВ 2
	REZ_3				:= 0			// РЕЗЕРВ 3
);

SETTS_DEF : TSetts:=
(
	// Температуры запуска приводов
	T_ZAP:=[180, 195, 210, 225, 220, 230, 230],

	// Время выгона массы в секундах
	TM_VIGON:=120,										

	// Флаг отключения звуковой сигнализации аварий
	otkl_alarm_zvuk:=FALSE,
	
	// Переменная для отключения ошибки "Превышение температуры одной из зон"
	otkl_h_temp:=FALSE,									

	// Переменная для отключения ошибки "Низкая температура одной из зон" 
	otkl_l_temp:=FALSE,
	
	// // Переменная для отключения контроля движения ТЯУ
	otkl_c_pulling:=FALSE,
	
	// Флаг выгона массы
	use_vigon:=TRUE,

	// Флаг использования бункера
	use_bunker:=TRUE,
	
	// Разрешить работу головки без разогрева (ТОЛЬКО ДЛЯ ОТЛАДКИ !!!)
	use_servo_without_temp:=FALSE,								

	// Разрешить работу шнека без разогрева (ТОЛЬКО ДЛЯ ОТЛАДКИ !!!)
	use_shnek_without_temp:=FALSE,

	// Флаг для условного включения зон 1-4
	CondEnableZones1_4:=TRUE,

	// Зона (5-1 .. 7-1), по которой управляется включение зон 1-4
	CondIZone:=6,

	// Значение 0-100 % от температуры уставки зоны (5-7), при превышении которой включаются зоны 1-4
	CondValue:=80,

	// Начальное положение (смещение) реперной точки относительно заднего концевика в 0.01 мм
	REP_MM:=-8.425,
	
	// Время выгона массы после вывода бункера в секундах
	TimeVigon:=180,
	
	// Длина заготовки в мм
	K_Length:=1265,
	
	// Температуры для автонастройки ПИД-регуляторов
	zd_temps:=[185, 200, 215, 230, 240, 240, 250]

);

END_VAR

VAR_GLOBAL

Nagrev				: TNagrev:=(T_Enables:=127);	// 127 = 1111111 b, то есть по умолчанию включены все 7 зон нагрева
Dvp					: TDVP;				// Переменные контроллера DVP
Asda				: TAsda;		// Переменные сервопривода
Chiller				: TChiller;		// Переменные Чиллера
Shnek				: TShnek;		// Переменные шнека
Pulling				: TPulling;		// Переменные тянущего устройства

frame_index			: BYTE:=0;		// Индекс закладки
frame_index_prev	: BYTE;			// Индекс предыдущей закладки
frame_index_reg		: BYTE;			// Индекс закладки настроек режима
frame_index_setts	: BYTE;			// Индекс закладки настроек системы
alarm_count			: INT;			// Число аварий и сообщений
ALARM				: BOOL;			// Флаг сигнализации 
ALARM_ZVUK			: BOOL;			// Флаг звуковой сигнализации
ALARM_PCHVS			: WORD;			// Общий контейнер сообщений от 2х частотников OWEN
ALARM_TEST			: BOOL;			// Тестовая авария
ALARM_MOVE			: BOOL:=TRUE;			// Флаг отсутствия движения заготовки
SBROS_AVARII		: BOOL;			// Общий импульс сброса сообщения
SBROS_AVARII_ASDA	: BOOL;			// Сигнал сброса сообщения только от сервопривода
SBROS_AVARII_RISING	: BOOL;			// Фронт импульса сброса сообщения

// Переменные для цвета окошек АКТУАЛЬНЫХ температур
clFillLowLow		: DWORD:=MERGE_RGB (128,128,255);	// Цвет заливки низкой величины
clFillLow			: DWORD:=MERGE_RGB (190,190,255);	// Цвет заливки пониженной величины
clFillMid			: DWORD:=MERGE_RGB (234,233,232);	// Цвет заливки нормальной величины
clFillHigh			: DWORD:=MERGE_RGB (255,190,190);	// Цвет заливки повышенной величины
clFillHighHigh		: DWORD:=MERGE_RGB (255,128,128);	// Цвет заливки высокой величины
clFillDisable		: DWORD:=MERGE_RGB (100,100,100);	// Цвет заливки недействительной величины

clFrameLowLow		: DWORD:=MERGE_RGB (0,0,255);		// Цвет фрейма низкой величины
clFrameLow			: DWORD:=MERGE_RGB (0,128,255);		// Цвет фрейма пониженной величины
clFrameMid			: DWORD:=MERGE_RGB (97,109,121);	// Цвет фрейма нормальной величины
clFrameHigh			: DWORD:=MERGE_RGB (255,128,0);		// Цвет фрейма высокой величины
clFrameHighHigh		: DWORD:=MERGE_RGB (255,0,0);		// Цвет фрейма повышенной величины
clFrameDisable		: DWORD:=MERGE_RGB (0,0,0);			// Цвет фрейма недействительной величины

// Переменные цвета кнопки
clFillBtnOn			: DWORD:=MERGE_RGB (128,255,128);	// Цвет заливки включенной кнопки ПУСК
clFillBtnOff		: DWORD:=MERGE_RGB (78,137,197);	// Цвет заливки разрешенной кнопки ПУСК
clFillBtnBreak		: DWORD:=MERGE_RGB (255,0,0);		// Цвет заливки запрещённой кнопки ПУСК

clFrameBtnOn		: DWORD:=MERGE_RGB (255,0,0);		// Цвет фрейма включенной кнопки ПУСК
clFrameBtnOff		: DWORD:=MERGE_RGB (128,255,128);	// Цвет фрейма разрешенной кнопки ПУСК
clFrameBtnBreak		: DWORD:=MERGE_RGB (128,255,128);	// Цвет фрейма аварийного состояния

FPS_FULL			: WORD;								// Суммарный FPS COM-портов

TEMPERS				: ARRAY [0..NUM_TEMPS-1] OF REAL;	// Результирующие уставки температур с учётом настроечных уставок для ПИД
PARAM_SET			: WORD;								// Переменная для активного набора параметров (1,2) управления ПЧВ ТЯУ

AddWriteCmd			: AddWriteCmd_FB;					// ФБ записи однократнй записи в COM-порт 

REG_TEMP			: TReg;								// Временный режим (для операций чтения и записи в файл)
pTargetReg			: POINTER TO TReg;					// Целевой режим (для операций чтения и записи в файл)
iMsgShowDlg			: WORD;								// Индекс сообщения в диалоге DlgShow;

parol_vvod			: WORD;								// Переменная для ввода пароля
b_n					: BOOL;								// Переменная блокировки по 

DELAY_ASDA			: PROCESS_DELAY_FB;

END_VAR

VAR_GLOBAL RETAIN

parol			: WORD:=13531;							// Переменная для пароля							
REG_W			: TReg:=REG_DEF;						// Текущий режим сервопривода
REG_ED			: TReg:=REG_DEF;						// Режим редактирования
Setts			: TSetts:=SETTS_DEF;					// Установки
// Archivate		: BOOL:=TRUE;							// Работать архиватору

END_VAR

// Device/Application/GVL_FILE
//{attribute 'qualified_only'}
VAR_GLOBAL CONSTANT

// Пути каталогов
DIR_USB_A			: STRING:='/mnt/ufs/media/sda1/';
DIR_USB_B			: STRING:='/mnt/ufs/media/sdb1/';
DIR_SD				: STRING:='/mnt/ufs/media/mmcblk0p1/';

// Имена файлов
FILE_NAME			: STRING:='saves_kar.dat';
TEMP_FILE_NAME		: STRING:='tempsaves_kar.dat';
OPTIONS_FILE_NAME	: STRING:='options_kar.dat';

TABLE_NUM_ROWS		: INT:=8;	// Число страниц в таблице режимов

END_VAR


VAR_GLOBAL

MMCMounted			: BOOL;			// Флаг монтирования MMC
EnableDrivers		: BOOL:=TRUE;	// Включены всегда
bUnmount			: BOOL;			// Импульс демонтирования SD карты
TBL					: TTable;		// Данные таблицы для выбора режима

Project				: TProject;

// Имя файла записи-чтения
FILENAME		: STRING:= CONCAT (DIR_SD, FILE_NAME);
TEMPFILE		: STRING:= CONCAT (DIR_SD, TEMP_FILE_NAME);
OPTIONSFILE		: STRING:= CONCAT (DIR_SD, OPTIONS_FILE_NAME);

END_VAR

// Device/Application/COM3_PRG
PROGRAM COM3_PRG
VAR CONSTANT
	COM3_TIME_OUT	: TIME:=T#800MS;
END_VAR

VAR
	Init			: BOOL:=FALSE;
	WR_REGS			: TRWRegs;			// Структура для записи в программе COM3
	RD_REGS			: TRWRegs;			// Структура для чтения в прогамме COM3
	COMPort3		: COM_SERVICE;			// ФБ настройки и открытия порта COM3
	Sets_COM		: COM_SETTINGS;
	Sets_COM_EX		: COM_SETTINGSex;
	CH_READ			: MB_RD_HOLD_REGS;		// ФБ чтения регистров чиллера
	CH_WRITE		: MB_WR_REGS;			// ФБ записи в регистр Чиллера
	abyBuffer		: ARRAY [0..255] OF BYTE;
	vWord			: WORD;
	vInt			: INT;
	xModule, I		: INT:=0;
	TM_FPS			: TON;
	tcount			: WORD;
	FPS				: WORD;
	Ready			: BOOL;						// Флаг готовности разового чтения или записи
	w_check			: BOOL;						// Переключатель при записи
	
	
END_VAR


IF NOT Init THEN
	// Настраиваем COM-порт
	Sets_COM.sPort:=3;
	Sets_COM.byStopBits:=SYS_ONESTOPBIT;
	Sets_COM.byParity:= SYS_EVENPARITY;
	Sets_COM.ulBaudrate:=SYS_BR_19200;
	Sets_COM.ulTimeout:=0;
	Sets_COM.ulBufferSize:=1024;
	Sets_COM_EX.byByteSize:=7;
	COMPort3 (Enable:=TRUE, Settings:=Sets_COM, Sets_EX:=Sets_COM_EX, Task:=OPEN_TSK);
	
	IF ComPort3.Ready THEN
		xModule:=10;
		Init:=TRUE;
	ELSE
		RETURN;
	END_IF

END_IF

//==========================================================		
// РАЗОВОЕ чтение 16 битных регистров при наличии в очереди 
//==========================================================
IF Ready AND RD_REGS.Count > 0 THEN
	// Чтение регистра 
	CH_READ (Enable:=ComPort3.Ready, Mode:=MB_ASCII, DevAddr:=RD_REGS.REGS[0].DevAdr, FirstAddr:=RD_REGS.REGS[0].RegAdr,
		Quantity:=RD_REGS.REGS[0].RegsCount, ComHandle:=ComPort3.handle, TimeOut:=COM3_TIME_OUT, Buffer:=abyBuffer);
		
	// Если чтение закончено
	IF CH_READ.Complete THEN
		//... и ошибки отсутствуют
		IF CH_READ.Exception = 0 THEN
			// Переписываем RegCount регистров начиная с нулевого
			FOR I:=0 TO RD_REGS.REGS[0].RegsCount-1 DO
				RD_REGS.REGS[0].pVals[I]:=WORD_FROM_BYTES (ADR (abyBuffer[I*2]));
			END_FOR
			tcount:=tcount + 1;
		END_IF
		
		CH_READ (Enable:=FALSE, Buffer:=abyBuffer);		// Завершаем опрос модуля
		QueuePopReg (ADR (RD_REGS));
	END_IF	

	RETURN;
END_IF 

//==========================================================		
// РАЗОВАЯ Запись массива 16 битных регистров при налмчии в очереди 
//==========================================================

IF Ready AND WR_REGS.Count > 0 THEN

	IF NOT w_check THEN
		// Записываем RegCount регистров начиная с нулевого.  (BYTES_FROM_WORD переставляет байты в слове)
		FOR I:=0 TO WR_REGS.REGS[0].RegsCount-1 DO
			vWord:=WR_REGS.REGS[0].pVals[I];
			BYTES_FROM_WORD (ADR (abyBuffer[I*2]), vWord );
		END_FOR
	END_IF
	
	CH_WRITE (Enable:=ComPort3.Ready, Mode:=MB_ASCII, DevAddr:=WR_REGS.REGS[0].DevAdr, FirstAddr:=WR_REGS.REGS[0].RegAdr,
		Quantity:=WR_REGS.REGS[0].RegsCount, ComHandle:=ComPort3.handle, TimeOut:=COM3_TIME_OUT, Buffer:=abyBuffer);
			
	w_check:=TRUE;
	IF CH_WRITE.Complete THEN
		// Если исключения отсутствуют
		IF CH_WRITE.Exception=0 THEN
			tcount:=tcount + 1;
		END_IF
		// Выключаем модуль записи
		CH_WRITE (Enable:=FALSE, Buffer:=abyBuffer);
		QueuePopReg (ADR (WR_REGS));
		w_check:=FALSE;
	END_IF
	
	RETURN;
END_IF	


CASE xModule OF
	//======================================================================================
10:	// ПОСТОЯННОЕ ЧТЕНИЕ требуемых регистров Чиллера (10 регистров)
	//======================================================================================
	Ready:=FALSE;
	CH_READ (Enable:=COMPort3.Ready, Mode:=MB_ASCII, DevAddr:=ADR_CHILLER, FirstAddr:=0, Quantity:=10, ComHandle:=COMPort3.handle, TimeOut:=COM3_TIME_OUT, Buffer:=aByBuffer);
	IF CH_READ.Complete THEN
		// Сбрасываем видимость
		Chiller.Connect:=FALSE;	
		IF CH_READ.Exception=0 THEN
			// .. и ошибки отсутствуют, то сразу же забираем буфер модуля
			Chiller.Connect:=TRUE;
			// Разбираем байты по переменным
			// 1. Текущая температура
			Chiller.T_ACTUAL:=INT_FROM_BYTES (ADR (aByBuffer[0])) * 0.1;
			// 2. Status flag
			Chiller.Status:=WORD_FROM_BYTES (ADR (aByBuffer[8]));
			// 3. Alarm flag 1
			Chiller.AlarmFlag1:=WORD_FROM_BYTES (ADR (aByBuffer[10]));
			// 4. Alarm flag 2
			Chiller.AlarmFlag2:=WORD_FROM_BYTES (ADR (aByBuffer[12]));
			// 5. Alarm flag 3
			Chiller.AlarmFlag3:=WORD_FROM_BYTES (ADR (aByBuffer[14]));
			// Авария Чиллера
			Chiller.AVAR:=Chiller.AlarmFlag1 <> 0 OR Chiller.AlarmFlag2 <> 0 OR Chiller.AlarmFlag3 <> 0;
			
			// 6. Status flag 2
			Chiller.Status_2:=WORD_FROM_BYTES (ADR (aByBuffer[18]));
			tcount:=tcount + 1;
		END_IF
		// Завершаем опрос чиллера
		CH_READ (Enable:=FALSE, Buffer:=aByBuffer);
		Ready:=TRUE;
		xModule:=10;					// Переход (?)

	END_IF

END_CASE	
	
// FPS for com3
TM_FPS (IN:=TRUE, PT:=T#1S);
IF TM_FPS.Q THEN
	TM_FPS (IN:=FALSE);
	FPS:=tcount;
	tcount:=0;
END_IF

END_PROGRAM

// Device/Application/SRC/WORD_FROM_BYTES
FUNCTION WORD_FROM_BYTES : WORD
VAR_INPUT
	pB : POINTER TO BYTE; 
END_VAR
VAR
	pB2	: POINTER TO BYTE;
END_VAR

pB2:=ADR (WORD_FROM_BYTES);
pB2[0]:=pB[1];
pB2[1]:=pB[0];

END_FUNCTION

// Device/Application/SRC/QueuePopReg
FUNCTION QueuePopReg : BOOL
VAR_INPUT
	pRegs	: POINTER TO TRWRegs;
END_VAR
VAR
	I: INT;
END_VAR

QueuePopReg:=FALSE;

IF pRegs^.Count > 0 THEN

	FOR I:=0 TO pRegs^.Count - 2 DO
		pRegs^.REGS [I]:=pRegs^.REGS [I+1];
	END_FOR

	pRegs^.Count:=pRegs^.Count-1;

END_IF

END_FUNCTION

// Device/Application/SRC/BYTES_FROM_WORD
FUNCTION BYTES_FROM_WORD : BOOL
VAR_INPUT
	pBytes	: POINTER TO BYTE;
	wWord	: WORD;
END_VAR
VAR
	pB		: POINTER TO BYTE;
END_VAR

BYTES_FROM_WORD:=TRUE;

pB:=ADR(wWord);
pBytes[0]:=pB[1];
pBytes[1]:=pB[0];

END_FUNCTION

// Device/Application/SRC/INT_FROM_BYTES
FUNCTION INT_FROM_BYTES : INT
VAR_INPUT
	pB : POINTER TO BYTE; 
END_VAR
VAR
	pB2	: POINTER TO BYTE;
END_VAR

pB2:=ADR (INT_FROM_BYTES);
pB2[0]:=pB[1];
pB2[1]:=pB[0];

END_FUNCTION

// Device/Application/CURRENT_PRG
PROGRAM CURRENT_PRG
VAR CONSTANT
	TimeSet			: WORD:=180;		// Время 3 мин на остановку шнека
END_VAR
VAR
	C_B				: BOOL:=FALSE;
	I				: INT;
	R_TRIG_NAGREV	: R_TRIG;
	R_TRIG_ZAP		: R_TRIG;
	R_TRIG_CH		: R_TRIG;
	F_TRIG_CH		: F_TRIG;
	R_TRIG_SH		: R_TRIG;
	F_TRIG_SH		: F_TRIG;
	R_TRIG_PL		: R_TRIG;
	F_TRIG_PL		: F_TRIG;
	R_TRIG_AL		: R_TRIG;
	R_TRIG_ZVUK		: R_TRIG;
	TON_AL			: TON;
	TON_AL_ASDA		: TON;
	STEP_R			: INT:=0;		
	R_AL			: R_TRIG;
	u_chil_old		: REAL;
	qm_old			: REAL;
	speed_old		: REAL;
	TP_MASS			: TP;
	F_TR_MASS		: F_TRIG;
	R_TRIG_0		: R_TRIG;
	TON_RD_PID		: TON;
	TON_WR_PID		: TON;
	TON_UNMOUNT		: TON;
	F_RD_PID		: F_TRIG;
	R_WR_PID		: R_TRIG;
	pid_index_old	: WORD:=255;
	NASOS_TOF		: TOF;
	VIGON_BLK		: BLINK;
	Vigon			: BOOL;		// Флаг выгона массы
	ShowDialog		: VU.FbOpenDialog;
	bShowDialog		: BOOL;
	TON_0			: TON;
	TON_1			: TON;
	ConfirmSaveAsDialog 	: VU.FbOpenDialog;
	bConfirmSaveAsDialog	: BOOL;
	
	ShnekPusk			: BOOL;
	
	
END_VAR


//===============================================================================================================
// Блокировка по паролю
//===============================================================================================================
b_n:=parol <> parol_vvod;

// Цвета окошек температур, критическое повышение и снижение
ButtonColor (ADR (Nagrev.Nagrev_on), ADR (C_B), ADR (Nagrev.NagrevFillColor), ADR (Nagrev.NagrevFrameColor));			// Отрисовка выключателя нагрева
ButtonColor (ADR (Shnek.Pusk), ADR (Shnek.Block), ADR (Shnek.FillColor), ADR (Shnek.FrameColor));						// Отрисовка выключателя шнека
ButtonColor (ADR (Asda.Pusk), ADR (Asda.Block), ADR (Asda.BtnFillColor), ADR (Asda.BtnFrameColor));						// Отрисовка выключателя головки
ButtonColor (ADR (Pulling.Pusk), ADR (Pulling.Block), ADR (Pulling.BtnFillColor), ADR (Pulling.BtnFrameColor));			// Отрисовка выключателя тянущего
ButtonColor (ADR (Chiller.Pusk), ADR (Chiller.Block), ADR (Chiller.BtnFillColor), ADR (Chiller.BtnFrameColor));			// Отрисовка выключателя ЧИЛЛЕРА

//===============================================================================================================
// УПРАВЛЕНИЕ БУНКЕРОМ
// Bunker_si = 0 - бункер введён
// Bunker_si = 1 - бункер выведён
//===============================================================================================================
IF NOT Dvp.Bunker_si THEN
	// Если бункер выведен
	Dvp.bunker_viveden_msg:=Nagrev.Nagrev_on;	
ELSE
	Dvp.bunker_viveden_msg:=FALSE;	
END_IF

//===============================================================================================================
// УПРАВЛЕНИЕ ЗАПУСКОМ 1-4 ЗОН
//===============================================================================================================
R_TRIG_NAGREV (CLK:=Nagrev.Nagrev_on AND Setts.CondEnableZones1_4);
IF R_TRIG_NAGREV.Q THEN
	// Если включили нагрев, то отключи 1-4 зоны
	Nagrev.T_Enables.0:=FALSE;
	Nagrev.T_Enables.1:=FALSE;
	Nagrev.T_Enables.2:=FALSE;
	Nagrev.T_Enables.3:=FALSE;
END_IF

// Обнаружение разогрева образцовой зоны и включение зон 1-4
R_TRIG_ZAP (CLK:=(Nagrev.T_Actuals[Setts.CondIZone-1] > REG_W.TEMPS[Setts.CondIZone-1] * Setts.CondValue / 100) AND Nagrev.Nagrev_on AND Setts.CondEnableZones1_4);
IF R_TRIG_ZAP.Q THEN
	Nagrev.T_Enables.0:=TRUE;
	Nagrev.T_Enables.1:=TRUE;
	Nagrev.T_Enables.2:=TRUE;
	Nagrev.T_Enables.3:=TRUE;
END_IF

//===============================================================================================================
// УПРАВЛЕНИЕ ВЫГОНОМ МАССЫ
//===============================================================================================================
// Если шнек работает (температура не ниже температур запуска приводов),
// то запустим таймер для выпуска массы
// Обнаруживаем спад его выхода и останавливаем систему (кроме ТЯУ, т.к. нужно "вытянуть" заготовку от головки) 
TP_MASS (IN:= NOT Dvp.Bunker_si AND Shnek.Pusk, PT:=DWORD_TO_TIME (Setts.TimeVigon * 1000));
F_TR_MASS (CLK:=TP_MASS.Q);
IF F_TR_MASS.Q THEN
	Nagrev.Nagrev_on:=FALSE;
	Asda.Pusk:=FALSE;
	Shnek.Pusk:=FALSE;
//	Pulling.Pusk:=FALSE;
END_IF
VIGON_BLK (ENABLE:=TP_MASS.Q, TIMELOW:=T#500MS, TIMEHIGH:=T#500MS);
Vigon:=VIGON_BLK.OUT AND TP_MASS.Q;

//================================================================================================================
// Остановка тянущего устроиства, головки и шнека при наезде на дальний концевик каретки - флаг ошибки E_BITS_si.6
//================================================================================================================
IF Dvp.E_BITS_si.6 THEN
	Asda.Pusk:=FALSE;
	Shnek.Pusk:=FALSE;
	Pulling.Pusk:=FALSE;
END_IF
//===============================================================================================================
// УПРАВЛЕНИЕ НАГРЕВОМ
//===============================================================================================================
GET_SET_TEMPERS ();				// Получить задания для температур
ProcessTempers ();

//===============================================================================================================
// ЧИЛЛЕР И НАСОС
//===============================================================================================================
// Блокировка включения Чиллера. Переменная Chiller.Block передаётся в функцию окраски окошка Чиллера в красный/зеленый/синий цвета
// Переменная введена из-за универсальности данной функции, а именно, передачи в неё адреса данной переменной
Chiller.Block:=(*NOT Chiller.Connect OR *) Chiller.AVAR;

IF Chiller.Connect THEN
	// Запись уставки в Чиллер
	IF REG_W.T_CHIL <> u_chil_old THEN
		AddWriteCmd (wcmd:=wcChiller_Ust);
		u_chil_old:=REG_W.T_CHIL;	
	END_IF

	// Включение Чиллера
	R_TRIG_CH (CLK:=Chiller.Pusk);
	IF R_TRIG_CH.Q THEN
		AddWriteCmd (wcmd:=wcChiller_Start);
	END_IF

	// Выключение Чиллера
	F_TRIG_CH (CLK:=Chiller.Pusk);
	IF F_TRIG_CH.Q THEN
		AddWriteCmd (wcmd:=wcChiller_Stop);
	END_IF

ELSE
//	Chiller.Pusk:=FALSE;
	u_chil_old:=0;
END_IF

IF Chiller.Block THEN
	Chiller.Pusk:=FALSE;
END_IF

// Включение насоса
// Затяжка работы насоса на 10 сек, т.к. чиллер после выключения работает около 30 сек
NASOS_TOF (IN:=Chiller.Pusk AND Chiller.Status.0 AND NOT Chiller.Status.1, PT:=T#30S); 			// См.документацию по Чиллеру (4.10.4 Status flag)
Dvp.Nasos_so:=NASOS_TOF.Q;

//===============================================================================================================
// ГОЛОВКА
//===============================================================================================================
// Выключение головки при срабатываеии блокировки
IF Asda.Block OR Asda.AllowManual THEN
	Asda.Pusk:=FALSE;
END_IF

//===============================================================================================================
// ШНЕК
//===============================================================================================================

// Выключение шнека по блокировке
IF Shnek.Block THEN
	Shnek.Pusk:=FALSE;
END_IF

// Запись уставки шнека
IF REG_W.Qm <> qm_old AND Shnek.Connect THEN
	AddWriteCmd(wcmd:=wcShnek_Ust);	// Передача уставки шнеку (см FB)
	qm_old:=REG_W.Qm;	
END_IF

// Включение шнека
R_TRIG_SH(CLK:=Shnek.Pusk);
IF R_TRIG_SH.Q THEN
	AddWriteCmd(wcmd:=wcShnek_Start);
END_IF

// Выключение шнека
F_TRIG_SH(CLK:=Shnek.Pusk);
IF F_TRIG_SH.Q THEN
	AddWriteCmd(wcmd:=wcShnek_Stop);
END_IF

// ДОБАВЛЕНО: При остановке заготовки и работающем шнеке НЕМЕДЛЕННО ОСТАНАВЛИВАМ ШНЕК
IF ALARM_MOVE AND ShnekPusk THEN
	ShnekPusk:=FALSE;
END_IF

// ДОБАВЛЕНО: Остновить шнек при аварии или превышения момента сервопривода головки через 3 сек
TON_1(IN:=(Asda.E_CODE.0 OR Asda.E_CODE.5)  AND ShnekPusk, PT:=T#3S);
IF TON_1.Q THEN
	ShnekPusk:=FALSE;
END_IF

//===============================================================================================================
// ТЯНУЩЕЕ УСТРОЙСТВО
//===============================================================================================================
// Запись уставки тянущего
IF REG_W.Speed <> speed_old AND Pulling.Connect THEN
	AddWriteCmd(wcmd:=wcPulling_Ust);
	speed_old:=REG_W.Speed;
END_IF

// Включение тянущего
R_TRIG_PL (CLK:=Pulling.Pusk);
IF R_TRIG_PL.Q THEN
	AddWriteCmd(wcmd:=wcPulling_Start);
END_IF

// Выключение тянущего 
F_TRIG_PL (CLK:=Pulling.Pusk);
IF F_TRIG_PL.Q THEN
	AddWriteCmd(wcmd:=wcPulling_Stop);
END_IF

//===============================================================================================================
// ПИД-РЕГУЛЯТОРЫ
//===============================================================================================================
// Установка зоны 1-7 и индекса 0-6 ПИД
Dvp.zone_index:=MAX (1, MIN (7, Dvp.zone_index));
Dvp.pid_index:=Dvp.zone_index-1;
 
// Установка текущего ПИД-регулятора и чтение его параметров на контроллере DVP
IF Dvp.pid_index <> pid_index_old THEN
	// Запись номера зоны 0-6 в Dvp
	QueuePushReg(ADR (COM1_PRG.WR_REGS), ADR_DVP, 4107, ADR (Dvp.pid_index), 1); 
	pid_index_old:=Dvp.pid_index;				// Сохраним
END_IF

// Формирование импульса чтения параметров ПИД-регулятора
// по ранее установленному номеру зоны нагрева внутри Dvp
// см. COM1_PRG - постоянная запись в Dvp импульс Dvp.pid_read
TON_RD_PID(IN:=Dvp.pid_read, PT:=T#1S);
IF TON_RD_PID.Q THEN
	Dvp.pid_read:=FALSE;
END_IF

// По спаду импульса чтения читаем из Dvp параметры ПИД 
F_RD_PID (CLK:=Dvp.pid_read);
IF F_RD_PID.Q THEN
	// Чтение 9 регистров из Dvp, начиная с адреса 4128 (см. Устройства.xls) с записью в текущую структуру ПИД
	QueuePushReg (ADR (COM1_PRG.RD_REGS), ADR_DVP, 4128, ADR (Dvp.Pids[Dvp.pid_index].formula),1);
	QueuePushReg (ADR (COM1_PRG.RD_REGS), ADR_DVP, 4129, ADR (Dvp.Pids[Dvp.pid_index].Kc_Kp),2);
	QueuePushReg (ADR (COM1_PRG.RD_REGS), ADR_DVP, 4131, ADR (Dvp.Pids[Dvp.pid_index].Ti_Ki),2);
	QueuePushReg (ADR (COM1_PRG.RD_REGS), ADR_DVP, 4133, ADR (Dvp.Pids[Dvp.pid_index].Td_Kd),2);
	QueuePushReg (ADR (COM1_PRG.RD_REGS), ADR_DVP, 4135, ADR (Dvp.Pids[Dvp.pid_index].Tf),2);
END_IF

// Формирование импульса чтения параметров ПИД-регулятора
// по ранее установленному номеру зоны нагрева внутри Dvp
// см. COM1_PRG - постоянная запись в Dvp импульс Dvp.pid_read
TON_WR_PID(IN:=Dvp.pid_write, PT:=T#1S);
IF TON_WR_PID.Q THEN
	Dvp.pid_write:=FALSE;
END_IF

// По спаду импульса записи пишем в Dvp параметры ПИД
R_WR_PID(CLK:=Dvp.pid_write);
IF R_WR_PID.Q THEN
	// Запись 9 регистров ПИД, начиная с адреса
	QueuePushReg (ADR (COM1_PRG.WR_REGS), ADR_DVP, 4128, ADR (Dvp.Pids[Dvp.pid_index].formula),1);
	QueuePushReg (ADR (COM1_PRG.WR_REGS), ADR_DVP, 4129, ADR (Dvp.Pids[Dvp.pid_index].Kc_Kp),2);
	QueuePushReg (ADR (COM1_PRG.WR_REGS), ADR_DVP, 4131, ADR (Dvp.Pids[Dvp.pid_index].Ti_Ki),2);
	QueuePushReg (ADR (COM1_PRG.WR_REGS), ADR_DVP, 4133, ADR (Dvp.Pids[Dvp.pid_index].Td_Kd),2);
	QueuePushReg (ADR (COM1_PRG.WR_REGS), ADR_DVP, 4135, ADR (Dvp.Pids[Dvp.pid_index].Tf),2);
 
END_IF

//===============================================================================================================
// "Температура достигнута"
//===============================================================================================================
// ТАКАЯ КОНСТРУКЦИЯ НЕ РАБОТАЕТ!!!
// R_TRIG_0 (CLK:=Dvp.temper_reached, Q=>Dvp.temper_reached_msg);
// Dvp.temper_reached_msg не устанавливается, может, потому, что используется в менеджере тревог ???
R_TRIG_0(CLK:=Nagrev.Temper_Reached);
IF R_TRIG_0.Q THEN
	Nagrev.Temper_Reached_msg:=TRUE;
END_IF
 
//===============================================================================================================
// ОБРАБОТКА ОШИБОК
//===============================================================================================================
// Формирование импульса сброса аварии 2 сек
TON_AL(IN:=SBROS_AVARII, PT:=T#2S);
IF TON_AL.Q THEN
	SBROS_AVARII:=FALSE;
END_IF

// Формирование РУЧНОГО импульса сброса аварии ASDA 2 сек
TON_AL_ASDA(IN:=SBROS_AVARII_ASDA, PT:=T#2S);
IF TON_AL_ASDA.Q THEN
	SBROS_AVARII_ASDA:=FALSE;
END_IF

// Формирование фронта импульса сброса аварии
R_AL (CLK:=SBROS_AVARII, Q=>SBROS_AVARII_RISING);

// Сброс ошибки
IF SBROS_AVARII_RISING THEN
	Nagrev.Temper_Reached_msg:=FALSE;
	Nagrev.E_temp_high:=FALSE;
	Nagrev.E_temp_low:=FALSE;
	ALARM:=FALSE;
	ALARM_ZVUK:=FALSE;
	ALARM_PCHVS:=0;						// Сборка частотников
END_IF

IF alarm_count < 0 THEN
	alarm_count:=0;				// При сбое
END_IF

// Обнаружение пропадания ошибок по спаду сигнала пропадания ошибок - отключение сигнализации и возврат окна
TON_0(IN:=alarm_count=0, PT:=T#300MS);
R_TRIG_AL (CLK:=TON_0.Q);
IF R_TRIG_AL.Q THEN
	IF frame_index = 1 THEN
		SET_FRAME_INDEX(frame_index_prev);	// Возвращаем окно
	END_IF	
	ALARM:=FALSE;
	ALARM_ZVUK:=FALSE;		// Отключение звука автоматически
END_IF

//===============================================================================================================
// ОБРАБОТКА СООБЩЕНИЙ ЭКСТРУДЕРА
//===============================================================================================================
IF TP_MASS.Q THEN
	Nagrev.text_id:=3;		// Система в режиме выгона массы
ELSIF NOT Nagrev.Temper_Reached AND Nagrev.Nagrev_on THEN
	Nagrev.text_id:=1;		// Система в режиме РАЗОГРЕВ
ELSIF Nagrev.Temper_reached AND Nagrev.Nagrev_on THEN
	Nagrev.text_id:=2;		// Система в РАБОЧЕМ режиме
ELSE
	Nagrev.text_id:=0;		// Система в ИСХОДНОМ состоянии
END_IF

//===============================================================================================================
// FPS
//===============================================================================================================
FPS_FULL:=COM1_PRG.FPS + COM2_PRG.FPS + COM3_PRG.FPS;

//===============================================================================================================
// ДИАЛОГИ ПАНЕЛИ ОПЕРАТОРА
//===============================================================================================================
// Диалог сообщения 
ShowDialog (itfClientFilter:=VU.Globals.AllClients, xExecute:=bShowDialog, sDialogName:='DlgShow', xModal:=TRUE);
IF ShowDialog.xDone THEN
	bShowDialog:=FALSE;
END_IF

// Диалог подтверждения записи по уже существующему имени
ConfirmSaveAsDialog (itfClientFilter:=VU.Globals.AllClients, xExecute:=bConfirmSaveAsDialog, sDialogName:='DlgConfirmSaveAs', xModal:=TRUE);
IF ConfirmSaveAsDialog.xDone THEN
	bConfirmSaveAsDialog:=FALSE;	// Сброс флага запуска диалога
END_IF

// Демонтирование SD карты
TON_UNMOUNT (IN:=bUnmount, PT:=T#1S);
IF TON_UNMOUNT.Q THEN
	bUnmount:=FALSE;	
END_IF

END_PROGRAM

// Device/Application/SRC/ButtonColor
FUNCTION ButtonColor : BOOL
VAR_INPUT
	pPusk		: POINTER TO BOOL;
	pBlock		: POINTER TO BOOL;
	pFillColor	: POINTER TO DWORD;
	pFrameColor	: POINTER TO DWORD;	
END_VAR
VAR
END_VAR


// Отрисовка выключателя тянущего
IF pBlock^ THEN
	pPusk^:=FALSE;
	pFillColor^:=clFillBtnBreak;
	pFrameColor^:=clFrameBtnBreak;
ELSIF pPusk^ THEN
	pFillColor^:=clFillBtnOn;
	pFrameColor^:=clFrameBtnOn;
ELSE	
	pFillColor^:=clFillBtnOff;
	pFrameColor^:=clFrameBtnOff;
END_IF

ButtonColor:=TRUE;

END_FUNCTION

// Device/Application/SRC/GET_SET_TEMPERS
FUNCTION GET_SET_TEMPERS : BOOL
VAR_INPUT
END_VAR
VAR
END_VAR


// Если выбор настроечных температур, то берём температуры из отдельного массива zd_temps
IF Dvp.zd_selector THEN
	TEMPERS[0]:=Setts.zd_temps[0];
	TEMPERS[1]:=Setts.zd_temps[1];
	TEMPERS[2]:=Setts.zd_temps[2];
	TEMPERS[3]:=Setts.zd_temps[3];
	TEMPERS[4]:=Setts.zd_temps[4];
	TEMPERS[5]:=Setts.zd_temps[5];
	TEMPERS[6]:=Setts.zd_temps[6];

ELSE
	// Иначе из массива температур режима
	TEMPERS[0]:=REG_W.TEMPS[0];
	TEMPERS[1]:=REG_W.TEMPS[1];
	TEMPERS[2]:=REG_W.TEMPS[2];
	TEMPERS[3]:=REG_W.TEMPS[3];
	TEMPERS[4]:=REG_W.TEMPS[4];
	TEMPERS[5]:=REG_W.TEMPS[5];
	TEMPERS[6]:=REG_W.TEMPS[6];

END_IF

GET_SET_TEMPERS:=TRUE;

END_FUNCTION

// Device/Application/SRC/ProcessTempers
PROGRAM ProcessTempers
VAR
	t_critical_low	: BOOL;
	t_critical_high	: BOOL;
	t_low			: BOOL;
	t_high			: BOOL;
	t_gol_block		: BOOL;	
	t_shnek_block	: BOOL;	
	t_vihod			: BOOL;

	I 				: BYTE;
	TP_H			: TP;
	TP_L			: TP;
	TRS_TRIGS		: ARRAY [0..NUM_TEMPS-2] OF RS;
	AUTO_TONS		: ARRAY [0..NUM_TEMPS-2] OF TON;
	
END_VAR

//===============================
// Функция разбора температур зон
// ==============================
t_critical_high:=FALSE;
t_vihod:=TRUE;
t_gol_block:=FALSE;
t_shnek_block:=FALSE;

FOR I:=0 TO NUM_TEMPS-1 DO

	// Цвета окошек текущих температур
	// Температурная зона отключена
	IF NOT EXTRACT (Nagrev.T_Enables, I) AND (I < NUM_TEMPS-1) THEN 
		Nagrev.FrameColors[I]:=clFrameDisable;
		Nagrev.FillColors[I]:=clFillDisable;
	
	// Температура намного ниже заданной
	ELSIF Nagrev.T_ACTUALS[I] < TEMPERS[I] - DT_MAXS[I] THEN
		Nagrev.FrameColors[I]:=clFrameLowLow;
		Nagrev.FillColors[I]:=clFillLowLow;

	// Температура намного выше заданной
	ELSIF Nagrev.T_Actuals[I] > TEMPERS[I] + DT_MAXS[I] THEN
		Nagrev.FrameColors[I]:=clFrameHighHigh;
		Nagrev.FillColors[I]:=clFillHighHigh;

	// Температура ниже заданной
	ELSIF Nagrev.T_Actuals[I] < TEMPERS[I] - DT_MINS[I] THEN
		Nagrev.FrameColors[I]:=clFrameLow;
		Nagrev.FillColors[I]:=clFillLow;
		
	// Температура выше заданной
	ELSIF Nagrev.T_Actuals[I] > TEMPERS[I] + DT_MINS[I] THEN
		Nagrev.FrameColors[I]:=clFrameHigh;
		Nagrev.FillColors[I]:=clFillHigh;
	// Температура в нормальных пределах
	ELSE
		Nagrev.FrameColors[I]:=clFrameMid;
		Nagrev.FillColors[I]:=clFillMid;	
	END_IF

	// Установка флага выхода на режим (температуру расплава игнорируем)
	TRS_TRIGS[I] (SET:=Nagrev.T_Actuals[I] >= TEMPERS[I] - DT_MINS[I], RESET1:=Nagrev.T_Actuals[I] < TEMPERS[I] - DT_MAXS[I]);
	IF NOT TRS_TRIGS[I].Q1 THEN
		t_vihod:=FALSE;
	END_IF

	// Разбор максимальных температур (i<=6)
	IF Nagrev.T_Actuals[I] > T_CRITICALS[I] THEN
		// Отключение зоны. Включение возможно только после снижения температуры зоны ниже критической и повторном включении флажка
		Nagrev.T_Enables:=DWORD_TO_WORD (PUTBIT (Nagrev.T_Enables, I, FALSE)); 
		t_critical_high:=TRUE;		// Включение критического флага
	END_IF
		
	// Разбор блокировки головки (i<=6)
	IF I>=4 THEN
		IF Nagrev.T_Actuals[I] < Setts.T_ZAP[I] THEN
			t_gol_block:=TRUE;
		END_IF
	END_IF
		
	// Разбор блокировки шнека (i<=6)
	IF Nagrev.T_Actuals[I] < Setts.T_ZAP[I] THEN
		t_shnek_block:=TRUE;
	END_IF
		
	//==========================================================
	// УПРАВЛЕНИЕ АВТОНАСТРОЙКОЙ ЗОН
	//==========================================================
	// Формирование импульса 3 сек для включения автонастройки ПИД-регуляторов зон 1-7
	// с помощью массива TON-триггеров. Соотвемствующие биты в слове Dvp.Auto_OUT включаются
	// кнопками включения автонастройки (i<=6)
	AUTO_TONS [I] (IN:=EXTRACT (Nagrev.Auto_OUT, I), PT:=T#3S);
	IF AUTO_TONS [I].Q THEN
		// Сброс бита по истечении времени 3 сек
		Nagrev.Auto_OUT:=DWORD_TO_BYTE (PUTBIT (Nagrev.Auto_OUT, I, FALSE));
		// Сброс таймера по истечении времени 3 сек				AUTO_TONS [I] (IN:=FALSE);				
	END_IF
END_FOR

// Установка флага выхода на режим
IF t_vihod THEN
	Nagrev.Temper_Reached:=TRUE;
END_IF

// При выключении нагрева блокируем флаг выхода на режим
IF NOT Nagrev.Nagrev_on THEN
	Nagrev.Temper_Reached:=FALSE;
END_IF

// В случае, если вышли на режим, проверяем температуры за границами DT_MAXS
// и ниже температур запуска приводов (данный цикл вынесен из цикла, который выше,
// т.к некорректно формировался Dvp.temper_reached
t_critical_low:=FALSE;
t_low:=FALSE;
t_high:=FALSE;
	
IF Nagrev.Temper_Reached THEN
	FOR I:=0 TO NUM_TEMPS-1 DO

		IF Nagrev.T_Actuals[I] < Setts.T_ZAP[I] THEN
			// Минимальная критическая температура - меньше температуры запуска приводов
			t_critical_low:=TRUE;
		END_IF
		
		IF Nagrev.T_Actuals[I] > TEMPERS[I] + DT_MAXS[I] THEN
			// Больше DT_MAXS		
			t_high:=TRUE;
			
		ELSIF Nagrev.T_Actuals[I] < TEMPERS[I] - DT_MAXS[I] THEN
			// Меньше DT_MAXS		
			t_low:=TRUE;
		END_IF
	END_FOR
END_IF

// Цвет окошка температуры масса
// Температура намного ниже заданной
IF  Nagrev.T_ActualMass < REG_W.T_MASS - DT_MASS_MAX THEN
	Nagrev.FrameColorMass:=clFrameLowLow;
	Nagrev.FillColorMass:=clFillLowLow;
	
// Температура намного ниже заданной
ELSIF Nagrev.T_ActualMass > REG_W.T_MASS + DT_MASS_MAX THEN
	Nagrev.FrameColorMass:=clFrameHighHigh;
	Nagrev.FillColorMass:=clFillHighHigh;
	
// Температура ниже заданной
ELSIF Nagrev.T_ActualMass < REG_W.T_MASS - DT_MASS_MIN THEN
	Nagrev.FrameColorMass:=clFrameLow;
	Nagrev.FillColorMass:=clFillLow;

// Температура выше заданной
ELSIF Nagrev.T_ActualMass > REG_W.T_MASS + DT_MASS_MIN THEN
	Nagrev.FrameColorMass:=clFrameHigh;
	Nagrev.FillColorMass:=clFillHigh;

// Температура в нормальных пределах
ELSE
	Nagrev.FrameColorMass:=clFrameMid;
	Nagrev.FillColorMass:=clFillMid;	
END_IF

// Цвет окошка температуры чиллера
// Температура намного ниже заданной
IF NOT Chiller.Status.0 (* Chiller.Pusk *) THEN
	Chiller.FrameColor:=clFrameDisable;
	Chiller.FillColor:=clFillDisable;

ELSIF  Chiller.T_ACTUAL < REG_W.T_CHIL - DT_CHIL_MAX THEN
	Chiller.FrameColor:=clFrameLowLow;
	Chiller.FillColor:=clFillLowLow;
	
// Температура намного ниже заданной
ELSIF Chiller.T_ACTUAL > REG_W.T_CHIL + DT_CHIL_MAX THEN
	Chiller.FrameColor:=clFrameHighHigh;
	Chiller.FillColor:=clFillHighHigh;
	
// Температура ниже заданной
ELSIF Chiller.T_ACTUAL < REG_W.T_CHIL - DT_CHIL_MIN THEN
	Chiller.FrameColor:=clFrameLow;
	Chiller.FillColor:=clFillLow;

// Температура выше заданной
ELSIF Chiller.T_ACTUAL > REG_W.T_CHIL + DT_CHIL_MIN THEN
	Chiller.FrameColor:=clFrameHigh;
	Chiller.FillColor:=clFillHigh;

// Температура в нормальных пределах
ELSE
	Chiller.FrameColor:=clFrameMid;
	Chiller.FillColor:=clFillMid;	
END_IF

// Добавим выходы за пределы по температуре чиллера
t_critical_high:=t_critical_high OR (Chiller.T_ACTUAL > T_CHIL_CRITICAL);

t_high:=t_high OR (Chiller.T_ACTUAL > (REG_W.T_CHIL + DT_CHIL_MAX));
t_low:=t_low OR (Chiller.T_ACTUAL < (REG_W.T_CHIL - DT_CHIL_MAX));


// Блокировка сервопривода по температуре
Asda.Block:=(t_gol_block AND NOT Setts.use_servo_without_temp) OR NOT Asda.Connect;

// Блокировка шнека по температуре
Shnek.Block:=(t_shnek_block AND NOT Setts.use_shnek_without_temp) OR NOT Shnek.Connect;

// Температура одной из зон ниже температуры запуска приводов
Nagrev.E_critical_low:=t_critical_low;
// Критическая температура одной из зон
Nagrev.E_critical_high:=t_critical_high;

// ФОРМИРОВАНИЕ и ДЕАКТИВАЦИЯ СООБЩЕНИЙ
// "Превышена температура одной из зон"
TP_H (IN:=SBROS_AVARII AND t_high, PT:=T#8M);
Nagrev.E_temp_high:=t_high AND Nagrev.Temper_Reached AND NOT Setts.otkl_h_temp AND NOT TP_H.Q;	

// "Низкая температура одной из зон"
TP_L (IN:=SBROS_AVARII AND t_low, PT:=T#8M);
Nagrev.E_temp_low:=t_low AND Nagrev.Temper_Reached AND NOT Setts.otkl_l_temp AND NOT TP_L.Q;

END_PROGRAM

// Device/Application/SRC/QueuePushReg
// Функция добавления записи значения адреса и значения регистра в очередь
FUNCTION QueuePushReg : BOOL
VAR_INPUT
	pRegs		: POINTER TO TRWRegs;
	DevAdr		: BYTE;
	RegAdr		: WORD;
	pValue		: POINTER TO WORD;
	RegCount	: BYTE; 
END_VAR
VAR
END_VAR


QueuePushReg:=FALSE;
IF pRegs^.Count < MAX_MODBUS_REGS THEN
	pRegs^.REGS[pRegs^.Count].DevAdr:=DevAdr;
	pRegs^.REGS[pRegs^.Count].RegAdr:=RegAdr;
	pRegs^.REGS[pRegs^.Count].pVals:= pValue;	
	pRegs^.REGS[pRegs^.Count].RegsCount:=RegCount;
	pRegs^.Count:=pRegs^.Count+1;
	QueuePushReg:=TRUE;
END_IF

END_FUNCTION

// Device/Application/COM1_PRG
PROGRAM COM1_PRG
VAR CONSTANT
	COM1_TIME_OUT	: TIME:=T#500MS;
	
END_VAR
VAR
	Init			: BOOL:=FALSE;
	WR_REGS			: TRWRegs;			// Структура для записи в программе COM1
	RD_REGS			: TRWRegs;			// Структура для чтения в прогамме COM1
	ComPort			: COM_SERVICE;		// Функциональный блок инициализации ком порта, запускается один раз
	Sets_COM		: COM_SETTINGS;
	Sets_COM_EX		: COM_SETTINGSex;
	RD_HOLD_REGS	: MB_RD_HOLD_REGS;			// Чтение из контроллера DVP-14SS2
	WR_HOLD_REGS	: MB_WR_REGS;				// Звапись в контроллер DVP-14SS2
	abyBuffer		: ARRAY [0..255] OF BYTE;
	xModule, I		: INT:=0;
	vWord			: WORD:=0;
	TM_FPS			: TON;
	tcount			: WORD;
	FPS				: WORD;
	Ready			: BOOL;						// Флаг готовности разового чтения или записи
	w_check			: BOOL;						// Переключатель при записи
	iTemp			: INT;
END_VAR



IF NOT Init THEN
	
	// Начальная инициализация уставок температур
	GET_SET_TEMPERS ();

	// Настраиваем COM-порт
	Sets_COM.sPort:=1;						// Номер порта (1 !!!!)
	Sets_COM.byStopBits:=SYS_TWOSTOPBITS;	// Стопбит: 1-1 бит,2-1.5 бит, 3-2 бита, по умолчанию 1-1 бит
	Sets_COM.byParity:=SYS_NOPARITY;		// Чётность: 0-нет,1-нечет,2-чет ???
	Sets_COM.ulBaudrate:=SYS_BR_115200;		// Скорость	
	Sets_COM.ulTimeout:=0;
	Sets_COM.ulBufferSize:=1024;
	Sets_COM_EX.byByteSize:=8;				// Количество информационных бит
	ComPort (Enable:=TRUE, Settings:=Sets_COM, Sets_Ex:=Sets_COM_EX, Task:=OPEN_TSK);

	IF ComPort.Ready THEN
		xModule:=10;
		Init:=TRUE;
	ELSE
		RETURN;
	END_IF

END_IF

//==========================================================		
// ПРИНУДИТЕЛЬНОЕ РАЗОВОЕ чтение 16 битных регистров при наличии в очереди 
//==========================================================
IF Ready AND RD_REGS.Count > 0 THEN
	// Чтение регистра 
	RD_HOLD_REGS (Enable:=ComPort.Ready, Mode:=MB_RTU, DevAddr:=RD_REGS.REGS[0].DevAdr, FirstAddr:=RD_REGS.REGS[0].RegAdr,
		Quantity:=RD_REGS.REGS[0].RegsCount, ComHandle:=ComPort.handle, TimeOut:=COM1_TIME_OUT, Buffer:=abyBuffer);
		
	// Если чтение закончено
	IF RD_HOLD_REGS.Complete THEN
		//... и ошибки отсутствуют
		IF RD_HOLD_REGS.Exception = 0 THEN
			// Переписываем RegCount регистров начиная с нулевого
			FOR I:=0 TO RD_REGS.REGS[0].RegsCount-1 DO
				RD_REGS.REGS[0].pVals[I]:=WORD_FROM_BYTES (ADR (abyBuffer[I*2]));
			END_FOR
			tcount:=tcount + 1;
		END_IF
		RD_HOLD_REGS (Enable:=FALSE, Buffer:=abyBuffer);	// Завершаем опрос модуля
		QueuePopReg (ADR (RD_REGS));
	END_IF	

	RETURN;
END_IF 
	
//==========================================================		
// ПРИНУДИТЕЛЬНАЯ РАЗОВАЯ Запись массива 16 битных регистров при наличии в очереди 
//==========================================================
IF Ready AND WR_REGS.Count > 0 THEN
	IF NOT w_check THEN
		// Записываем RegCount регистров начиная с нулевого.  (BYTES_FROM_WORD переставляет байты в слове)
		FOR I:=0 TO WR_REGS.REGS[0].RegsCount-1 DO
			vWord:=WR_REGS.REGS[0].pVals[I];
			BYTES_FROM_WORD (ADR (abyBuffer[I*2]), vWord );
		END_FOR
	END_IF
	
	WR_HOLD_REGS (Enable:=ComPort.Ready, Mode:=MB_RTU, DevAddr:=WR_REGS.REGS[0].DevAdr, FirstAddr:=WR_REGS.REGS[0].RegAdr,
		Quantity:=WR_REGS.REGS[0].RegsCount, ComHandle:=ComPort.handle, TimeOut:=COM1_TIME_OUT, Buffer:=abyBuffer);
	
	w_check:=TRUE;		
	IF WR_HOLD_REGS.Complete THEN
		tcount:=tcount + 1;
		WR_HOLD_REGS (Enable:=FALSE, Buffer:=abyBuffer);	// Выключаем модуль записи
		QueuePopReg (ADR (WR_REGS));
		w_check:=FALSE;		
	END_IF

	RETURN;		// Выход с сохранением xModule
END_IF	


CASE xModule OF
	
	//====================================================================================
10:	// ПОСТОЯННАЯ ЗАПИСЬ в DVP-14SS2 - 11 регистров D0-D10, начиная с адреса 4096(16#1000) 
	//====================================================================================
	Ready:=FALSE;
	IF NOT w_check THEN
		BYTES_FROM_WORD (ADR (abyBuffer[0]), REAL_TO_WORD (TEMPERS[0]*10.0));		// Уставка температуры зоны 1
		BYTES_FROM_WORD (ADR (abyBuffer[2]), REAL_TO_WORD (TEMPERS[1]*10.0));		// Уставка температуры зоны 2
		BYTES_FROM_WORD (ADR (abyBuffer[4]), REAL_TO_WORD (TEMPERS[2]*10.0));		// Уставка температуры зоны 3
		BYTES_FROM_WORD (ADR (abyBuffer[6]), REAL_TO_WORD (TEMPERS[3]*10.0));		// Уставка температуры зоны 4
		BYTES_FROM_WORD (ADR (abyBuffer[8]), REAL_TO_WORD (TEMPERS[4]*10.0));		// Уставка температуры зоны 5
		BYTES_FROM_WORD (ADR (abyBuffer[10]), REAL_TO_WORD (TEMPERS[5]*10.0));		// Уставка температуры зоны 6
		BYTES_FROM_WORD (ADR (abyBuffer[12]), REAL_TO_WORD (TEMPERS[6]*10.0));		// Уставка температуры зоны 7
		BYTES_FROM_WORD (ADR (abyBuffer[14]), REAL_TO_WORD (REG_W.Speed * 10));		// Скорость движения в процентах
		BYTES_FROM_WORD (ADR (abyBuffer[16]), REAL_TO_WORD (Setts.K_Length * 10));	// Длина заготовки в 0.1 мм

		vWord.0:= Nagrev.T_Enables.0 AND Nagrev.Nagrev_on;
		vWord.1:= Nagrev.T_Enables.1 AND Nagrev.Nagrev_on;
		vWord.2:= Nagrev.T_Enables.2 AND Nagrev.Nagrev_on;
		vWord.3:= Nagrev.T_Enables.3 AND Nagrev.Nagrev_on;
		vWord.4:= Nagrev.T_Enables.4 AND Nagrev.Nagrev_on;
		vWord.5:= Nagrev.T_Enables.5 AND Nagrev.Nagrev_on;
		vWord.6:= Nagrev.T_Enables.6 AND Nagrev.Nagrev_on;
		vWord.7:= 0;

		vWord.8:= Nagrev.Auto_OUT.0; 
		vWord.9:= Nagrev.Auto_OUT.1; 
		vWord.10:=Nagrev.Auto_OUT.2; 
		vWord.11:=Nagrev.Auto_OUT.3; 
		vWord.12:=Nagrev.Auto_OUT.4; 
		vWord.13:=Nagrev.Auto_OUT.5; 
		vWord.14:=Nagrev.Auto_OUT.6; 
		vWord.15:= 0;

		BYTES_FROM_WORD (ADR (abyBuffer[18]), vWord);			
	
		// Управляющие биты
		vWord:=0;												// Управляющие биты
		vWord.0:=SBROS_AVARII;									// Импульс сброса аварии
		vWord.1:=Dvp.Nasos_so OR Dvp.Nasos_OTL;					// Сигнал включения насоса
		vWord.2:=ALARM;											// Сигнал аварийной сигнализации
		vWord.3:=Setts.otkl_alarm_zvuk OR NOT ALARM_ZVUK;		// Сигнал отключения звуковой сигнализации (1 - отлючение звука)
		vWord.4:=Pulling.Pusk;									// Сигнал включения тянущего устройства (вспомогательный)
		vWord.5:=Dvp.pid_read;									// Импульс операции для чтения ПИД внутри Dvp
		vWord.6:=Dvp.pid_write;									// Импульс операции для записи ПИД внутри Dvp  
		vWord.7:=Setts.otkl_c_pulling;							// Отключение контроля движения ТЯУ
		BYTES_FROM_WORD (ADR (abyBuffer[20]), vWord);			// Управляющие биты
	END_IF

	WR_HOLD_REGS (Enable:=ComPort.Ready, Mode:=MB_RTU, DevAddr:=ADR_DVP, FirstAddr:=16#1000, Quantity:=11, ComHandle:=ComPort.handle, TimeOut:=COM1_TIME_OUT, Buffer:=abyBuffer);

	w_check:=TRUE;
	IF WR_HOLD_REGS.Complete THEN
		tcount:=tcount + 1;
		WR_HOLD_REGS (Enable:=FALSE, Buffer:=abyBuffer);		// Выключаем модуль записи
		Ready:=TRUE;
		w_check:=FALSE;
		xModule:=20;											// Переходим далее
	END_IF

	//======================================================================================
20:	// ПОСТОЯННОЕ ЧТЕНИЕ из DVP-14SS2 - 11 регистров D16-D26, начиная с адреса 4112(16#1010) 
	//======================================================================================
	Ready:=FALSE;
	RD_HOLD_REGS (Enable:=ComPort.Ready, Mode:=MB_RTU, DevAddr:=ADR_DVP, FirstAddr:=16#1010, Quantity:=11, ComHandle:=ComPort.handle, TimeOut:=COM1_TIME_OUT, Buffer:=abyBuffer);
	IF RD_HOLD_REGS.Complete THEN
		// Сбрасываем соединение
		Dvp.Connect:=FALSE;
		IF RD_HOLD_REGS.Exception = 0 THEN
			//... и ошибки отсутствуют
			Dvp.Connect:=TRUE; // Присваиваем
			// Температуры
			Nagrev.T_Actuals[0]:=WORD_FROM_BYTES(ADR(abyBuffer[0])) * 0.1;	// Температура зоны 1
			Nagrev.T_Actuals[1]:=WORD_FROM_BYTES(ADR(abyBuffer[2])) * 0.1;	// Температура зоны 1
			Nagrev.T_Actuals[2]:=WORD_FROM_BYTES(ADR(abyBuffer[4])) * 0.1;	// Температура зоны 1
			Nagrev.T_Actuals[3]:=WORD_FROM_BYTES(ADR(abyBuffer[6])) * 0.1;	// Температура зоны 1
			Nagrev.T_Actuals[4]:=WORD_FROM_BYTES(ADR(abyBuffer[8])) * 0.1;	// Температура зоны 1
			Nagrev.T_Actuals[5]:=WORD_FROM_BYTES(ADR(abyBuffer[10])) * 0.1;	// Температура зоны 1
			Nagrev.T_Actuals[6]:=WORD_FROM_BYTES(ADR(abyBuffer[12])) * 0.1;	// Температура зоны 1
			Nagrev.T_ActualMass:=WORD_FROM_BYTES(ADR(abyBuffer[14])) * 0.1;	// Температура расплава

			// Биты ошибок
			Dvp.E_BITS_si:=WORD_FROM_BYTES(ADR(abyBuffer[16]));
			ALARM_MOVE:=Dvp.E_BITS_si.10;	// Авария отсутствия движения заготовки ТЯУ
			Dvp.Encoder:=Dvp.E_BITS_si.11;	// Флаг вращения энкодера

			// Состояния каналов			
			vWord:= WORD_FROM_BYTES (ADR (abyBuffer[18]));
			Nagrev.T_Enables_si.0:=vWord.0;
			Nagrev.T_Enables_si.1:=vWord.1;
			Nagrev.T_Enables_si.2:=vWord.2;
			Nagrev.T_Enables_si.3:=vWord.3;
			Nagrev.T_Enables_si.4:=vWord.4;
			Nagrev.T_Enables_si.5:=vWord.5;
			Nagrev.T_Enables_si.6:=vWord.6;

			// Фиксация завершения самонастроек каналов нагрева
			Nagrev.Auto_IN.0:=vWord.8;		
			Nagrev.Auto_IN.1:=vWord.9;
			Nagrev.Auto_IN.2:=vWord.10;
			Nagrev.Auto_IN.3:=vWord.11;
			Nagrev.Auto_IN.4:=vWord.12;
			Nagrev.Auto_IN.5:=vWord.13;
			Nagrev.Auto_IN.6:=vWord.14;

			// Управляющие биты
			vWord:=WORD_FROM_BYTES (ADR (abyBuffer[20]));
			Dvp.Uroven_s_si	:= vWord.0;		// Датчик уровня сырья в бункере
			Dvp.Bunker_si	:= vWord.1;		// Положение бункера 0-выведен, 1-введён
			Dvp.PVozd_si	:= vWord.2;		// Давление воздуха
			Dvp.KarIsx_si	:= vWord.3;		// Датчик исходного положения каркаса
			Dvp.KarRab_si	:= vWord.4;		// Датчик рабочего положения каркаса
			Dvp.ZazhIsx_si	:= vWord.5;		// Датчик исходного положения зажима
			Dvp.Uroven_w_si	:= vWord.6;		// Датчик уровня воды в баке
			Dvp.KnifeIsx_si	:= vWord.7;		// Датчик исходного положения ножа
			Dvp.KnifeRab_si	:= vWord.8;		// Датчик рабочего положения ножа

			Dvp.Nasos_si		:= vWord.9;		// Реле включения насоса
			Dvp.Karet_si		:= vWord.10;	// Пневмоцилиндр каретки
			Dvp.Zazh_si			:= vWord.11;	// Пневмоцилиндр зажима
			Dvp.Knife_si		:= vWord.12;	// Пневмоцидиндр ножа
			Dvp.F_OTR_si		:= vWord.13;	// Импульс отрезки заготовки
			Dvp.STOP_MANUAL_si	:= vWord.14;	// Сигнал аварийного останова от кнопки СТОП (ИНВЕРСНЫЙ)

			tcount:=tcount + 1;
		END_IF
		// Завершаем опрос модуля
		RD_HOLD_REGS (Enable:=FALSE, Buffer:=abyBuffer);	
		Ready:=TRUE;
		xModule:=25;
	END_IF

	//===================================================================================================================
25:	// ПОСТОЯННОЕ ЧТЕНИЕ из ASDA_A2 всех необходимых параметров одной командой чтения
	// с помощью отображения (через параметры P0-25 - P0-32, P0-35 - P0-42)
	// Последовательность регистров задаётся в параметрах P0-35 - P0-42, Чтение значений - P0-25 - P0-32
	// Задана последовательность:
	// 1,2. P2-30, P3-06 отображаются через loword и highword соответственно параметра P0-25, задаются в параметре P0-35
	// 3,4. P4-07, P0-46 отображаются через loword и highword соответственно параметра P0-26, задаются в параметре P0-36
	// 5,6. Р5-07, P0-01 отображаются через loword и highword соответственно параметра P0-27, задаются в параметре P0-37
	// 7. P0-09 - монитор состояния 1 для "Входная команда момента %". В параметре P0-17 д.б. записано число 11.
	
	// P0-09 отображается через loword и highword P0-28 (как 32-битное), задаётся в параметре P0-38 *)
 
	// Установить параметр P3-07 = 4 (Задержка ответа от сервопривода 2 мс, при задержке 0 мс возникают ошибки при чтении
	// При чтении начальный адрес - 16#0032 - регистр P0-25, число регистров 6+2=8.
	// Кроме того установить в параметр установить параметр P3-07 = 4 (Зажержка ответа от сервопривода 2 мс, при задержке 0 мс возникают ошибки при чтении
	//===================================================================================================================
	Ready:=FALSE;
	RD_HOLD_REGS (Enable:=ComPort.Ready, Mode:=MB_RTU, DevAddr:=ADR_ASDA, FirstAddr:=16#0032, Quantity:=8, ComHandle:=ComPort.handle, TimeOut:=COM1_TIME_OUT, Buffer:=abyBuffer);
	IF RD_HOLD_REGS.Complete THEN
		//... если закончили чтение
		Asda.Connect:=FALSE;
		IF RD_HOLD_REGS.Exception = 0 THEN
			// ... И отсутствуют ошибки
			Asda.Connect:=TRUE;		// Присваиваем
			Asda.P2_30:=WORD_FROM_BYTES (ADR (abyBuffer[0]));		// Чтение P2-30
			Asda.P3_06:=WORD_FROM_BYTES (ADR (abyBuffer[2]));		// Чтение P3-06
			Asda.P4_07:=WORD_FROM_BYTES (ADR (abyBuffer[4]));		// Чтение P4-07
			Asda.P0_46:=WORD_FROM_BYTES (ADR (abyBuffer[6]));		// Чтение P0-46
			Asda.P5_07:=WORD_FROM_BYTES (ADR (abyBuffer[8]));		// Чтение P5-07
			Asda.P0_01:=WORD_FROM_BYTES (ADR (abyBuffer[10]));		// Чтение P0-01
			Asda.E_ALARM:=BCD_TO_WORD (Asda.P0_01);					// Конвертируем BCD в WORD

			iTemp:=INT_FROM_BYTES (ADR (abyBuffer[12]));			// Хотя передаётся число DWORD Читаем только младший байт
			Asda.TorqueMin:=MIN (Asda.TorqueMin, iTemp);
			Asda.TorqueMax:=MAX (Asda.TorqueMax, iTemp);
			Asda.Torque:=iTemp;
			tcount:=tcount + 1;
		END_IF
		RD_HOLD_REGS (Enable:=FALSE, Buffer:=abyBuffer);		// Завершаем опрос модуля
		Ready:=TRUE;
		xModule:=10;				// На начало
	END_IF
	
(*				
	//=======================================================================================================================
30:	// ПОСТОЯННОЕ ЧТЕНИЕ из ASDA_A2: параметр Р5-07 - СОСТОЯНИЕ ВЫПОЛНЕНИЯ КОМАНДЫ PR 
	// Установить параметр P3-07 = 4 (Зажержка ответа от сервопривода 2 мс, при задержке 0 мс возникают ошибки при чтении
	//=======================================================================================================================
	Ready:=FALSE;
	RD_HOLD_REGS (Enable:=ComPort.Ready, Mode:=MB_RTU, DevAddr:=ADR_ASDA, FirstAddr:=16#050E, Quantity:=1, ComHandle:=ComPort.handle, TimeOut:=COM1_TIME_OUT, Buffer:=abyBuffer);
	IF RD_HOLD_REGS.Complete THEN
		//... и ошибки отсутствуют
		Asda.Connect:=FALSE;
	
		IF RD_HOLD_REGS.Exception = 0 THEN
			Asda.Connect:=TRUE;	// Присваиваем
			Asda.P5_07:=WORD_FROM_BYTES(ADR(abyBuffer[0]));		// Чтение P5-07
			tcount:=tcount + 1;
		END_IF

		RD_HOLD_REGS (Enable:=FALSE, Buffer:=abyBuffer);		// Завершаем опрос модуля
		Ready:=TRUE;
		xModule:=40;
	END_IF

	//=======================================================================================================================
40:	// ПОСТОЯННОЕ ЧТЕНИЕ из ASDA_A2 привода пилы: параметр Р4-07 - СОСТОЯНИЕ ДИСКРЕТНЫХ ВХОДОВ, адрес регистра 16#040E 
	//=======================================================================================================================
	Ready:=FALSE;
	RD_HOLD_REGS (Enable:=ComPort.Ready, Mode:=MB_RTU, DevAddr:=ADR_ASDA, FirstAddr:=16#040E, Quantity:=1, ComHandle:=ComPort.handle, TimeOut:=COM1_TIME_OUT, Buffer:=abyBuffer);
	IF RD_HOLD_REGS.Complete THEN
		//... и ошибки отсутствуют
		IF RD_HOLD_REGS.Exception = 0 THEN
			Asda.P4_07:=WORD_FROM_BYTES(ADR(abyBuffer[0]));		// Чтение P4-07 (состояние дискретных выходов)
			tcount:=tcount + 1;
		END_IF
		
		RD_HOLD_REGS (Enable:=FALSE, Buffer:=abyBuffer);		// Завершаем опрос модуля
		Ready:=TRUE;
		xModule:=50;
	END_IF
	
	//=======================================================================================================================
50:	// ПОСТОЯННОЕ ЧТЕНИЕ из ASDA_A2: параметр Р0-46 - СОСТОЯНИЕ ДИСКРЕТНЫХ ВЫХОДОВ, адрес регистра 16#005C 
	//=======================================================================================================================
	Ready:=FALSE;
	RD_HOLD_REGS (Enable:=ComPort.Ready, Mode:=MB_RTU, DevAddr:=ADR_ASDA, FirstAddr:=16#005C, Quantity:=1, ComHandle:=ComPort.handle, TimeOut:=COM1_TIME_OUT, Buffer:=abyBuffer);
	IF RD_HOLD_REGS.Complete THEN
		//... и ошибки отсутствуют
		IF RD_HOLD_REGS.Exception = 0 THEN
			Asda.P0_46:=WORD_FROM_BYTES(ADR(abyBuffer));		// Чтение P0-46
			tcount:=tcount + 1;
		END_IF
		
		RD_HOLD_REGS (Enable:=FALSE, Buffer:=abyBuffer);		// Завершаем опрос модуля
		Ready:=TRUE;
		xModule:=10;				// На начало
	END_IF
*)

END_CASE

// FPS for com1
TM_FPS (IN:=TRUE, PT:=T#1S);
IF TM_FPS.Q THEN
	TM_FPS (IN:=FALSE);
	FPS:=tcount;
	tcount:=0;
END_IF

END_PROGRAM

// Device/Application/SRC_AUX/LoWord
FUNCTION LoWord : WORD
VAR_INPUT
	dValue	: DINT;
END_VAR
VAR
	pW		: POINTER TO WORD;
END_VAR

pW:= ADR (dValue);
LoWord:=pW[0];

END_FUNCTION

// Device/Application/SRC/SET_FRAME_INDEX
FUNCTION SET_FRAME_INDEX : BOOL
VAR_INPUT
	Index : BYTE;
END_VAR
VAR
END_VAR
VAR // added by the converter: edge detectors and wires of the graphical bodies
    _w1 : BOOL;
    _w2 : ANY;
    _w3 : BYTE;
END_VAR

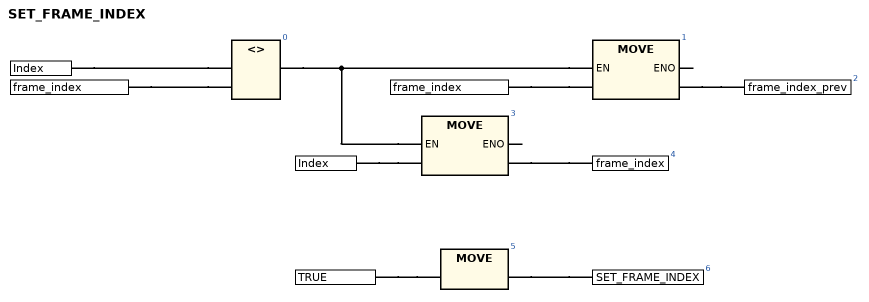
_w1 := Index <> frame_index;
IF _w1 THEN _w2 := frame_index; END_IF
frame_index_prev := _w2;
IF _w1 THEN _w3 := Index; END_IF
frame_index := _w3;
SET_FRAME_INDEX := TRUE;

END_FUNCTION

// Device/Application/COM2_PRG
PROGRAM COM2_PRG
VAR CONSTANT
	COM2_TIME_OUT	: TIME:=T#500MS;
END_VAR
VAR
	Init			: BOOL:=FALSE;
	WR_REGS			: TRWRegs;			// Структура для записи в программе COM3
	RD_REGS			: TRWRegs;			// Структура для чтения в прогамме COM3
	ComPort2		: COM_SERVICE;						// Функциональный блок инициализации ком порта, запускается один раз
	Sets_COM		: COM_SETTINGS;
	Sets_COM_EX		: COM_SETTINGSex;
	RD_HOLD_REGS	: MB_RD_HOLD_REGS;			// Чтение из контроллера DVP-14SS2
	WR_HOLD_REGS	: MB_WR_REGS;				// Звапись в контроллер DVP-14SS2
	abyBuffer		: ARRAY [0..255] OF BYTE;
	xModule, I		: INT:=0;
	vWord			: WORD;
	TM_FPS			: TON;
	tcount			: WORD;
	FPS				: WORD;
	Ready			: BOOL;						// Флаг готовности разового чтения или записи
	w_check			: BOOL;						// Переключатель при записи
END_VAR


IF NOT Init THEN
	// Настраиваем COM-порт
	Sets_COM.sPort:=2;						// Номер порта (2 - COM-порт для взаимодействия с двумя частотными преобразователями !!!!)
	Sets_COM.byStopBits:=SYS_ONESTOPBIT;	// Стопбит: 1-1 бит,2-1.5 бит, 3-2 бита, по умолчанию 1-1 бит
	Sets_COM.byParity:=SYS_NOPARITY;		// Чётность: 0-нет,1-нечет,2-чет ???
	Sets_COM.ulBaudrate:=SYS_BR_38400;		// Скорость	
	Sets_COM.ulTimeout:=0;
	Sets_COM.ulBufferSize:=1024;
	Sets_COM_EX.byByteSize:=8;				// Количество информационных бит
	ComPort2 (Enable:=TRUE, Settings:=Sets_COM, Sets_Ex:=Sets_COM_EX, Task:=OPEN_TSK);

	IF ComPort2.Ready THEN
		xModule:=10;
		Init:=TRUE;
	ELSE
		RETURN;
	END_IF
END_IF

//========================================================================		
// ПРИНУДИТЕЛЬНОЕ РАЗОВОЕ чтение 16 битных регистров при наличии в очереди 
//========================================================================
IF Ready AND RD_REGS.Count > 0 THEN
	// Чтение регистра 
	RD_HOLD_REGS (Enable:=ComPort2.Ready, Mode:=MB_RTU, DevAddr:=RD_REGS.REGS[0].DevAdr, FirstAddr:=RD_REGS.REGS[0].RegAdr,
		Quantity:=RD_REGS.REGS[0].RegsCount, ComHandle:=ComPort2.handle, TimeOut:=COM2_TIME_OUT, Buffer:=abyBuffer);
	// Если чтение закончено
	IF RD_HOLD_REGS.Complete THEN
		//... и ошибки отсутствуют
		IF RD_HOLD_REGS.Exception = 0 THEN
			// Переписываем RegCount регистров начиная с нулевого
			FOR I:=0 TO RD_REGS.REGS[0].RegsCount-1 DO
				RD_REGS.REGS[0].pVals[I]:=WORD_FROM_BYTES (ADR (abyBuffer[I*2]));
			END_FOR
			tcount:=tcount + 1;
		END_IF
		RD_HOLD_REGS (Enable:=FALSE, Buffer:=abyBuffer);		// Завершаем опрос модуля
		QueuePopReg (ADR (RD_REGS));
	END_IF	
	RETURN;													// Выход с сохранением xModule
END_IF		

//================================================================================		
// ПРИНУДИТЕЛЬНАЯ РАЗОВАЯ Запись массива 16 битных регистров при наличии в очереди 
//================================================================================
IF Ready AND WR_REGS.Count > 0 THEN

	IF NOT w_check THEN
		// Записываем RegCount регистров начиная с нулевого.  (BYTES_FROM_WORD переставляет байты в слове)
		FOR I:=0 TO WR_REGS.REGS[0].RegsCount-1 DO
			vWord:=WR_REGS.REGS[0].pVals[I];
			BYTES_FROM_WORD (ADR (abyBuffer[I*2]), vWord );
		END_FOR
	END_IF
	
	WR_HOLD_REGS (Enable:=ComPort2.Ready, Mode:=MB_RTU, DevAddr:=WR_REGS.REGS[0].DevAdr, FirstAddr:=WR_REGS.REGS[0].RegAdr,
		Quantity:=WR_REGS.REGS[0].RegsCount, ComHandle:=ComPort2.handle, TimeOut:=COM2_TIME_OUT, Buffer:=abyBuffer);
			
	w_check:=TRUE;
	IF WR_HOLD_REGS.Complete THEN
		tcount:=tcount + 1;
		WR_HOLD_REGS (Enable:=FALSE, Buffer:=abyBuffer);
		QueuePopReg (ADR (WR_REGS));
		w_check:=FALSE;
	END_IF	
	RETURN;													// Выход с сохранением xModule
END_IF	


CASE xModule OF
	//======================================================================================
10:	// Постоянное чтение регистра слова состояния STW привода шнека 
	//======================================================================================
	Ready:=FALSE;
	RD_HOLD_REGS (Enable:=ComPort2.Ready, Mode:=MB_RTU, DevAddr:=ADR_SHNEK, FirstAddr:=16#C417, Quantity:=1, ComHandle:=ComPort2.handle, TimeOut:=COM2_TIME_OUT, Buffer:=abyBuffer);
	IF RD_HOLD_REGS.Complete THEN
		// Сбрасываем соединение
		Shnek.Connect:=FALSE;
		IF RD_HOLD_REGS.Exception = 0 THEN
			//... и ошибки отсутствуют
			Shnek.Connect:=TRUE; // Присваиваем
			Shnek.STW:=WORD_FROM_BYTES (ADR (abyBuffer[0]));	// Слово состояния шнека
			
			IF Shnek.STW.3 THEN ALARM_PCHVS.0:=TRUE; END_IF
			IF Shnek.STW.7 THEN ALARM_PCHVS.1:=TRUE; END_IF
			IF Shnek.STW.13 THEN ALARM_PCHVS.2:=TRUE; END_IF
			IF Shnek.STW.14 THEN ALARM_PCHVS.3:=TRUE; END_IF
			IF Shnek.STW.15 THEN ALARM_PCHVS.4:=TRUE; END_IF
				
			tcount:=tcount + 1;
		END_IF
		// Завершаем опрос модуля
		RD_HOLD_REGS (Enable:=FALSE, Buffer:=abyBuffer);
		Ready:=TRUE;
		xModule:=20;
	END_IF

	//======================================================================================
20:	// Постоянное чтение регистра основного текущего значения MAV привода шнека 
	//======================================================================================
	Ready:=FALSE;
	RD_HOLD_REGS (Enable:=ComPort2.Ready, Mode:=MB_RTU, DevAddr:=ADR_SHNEK, FirstAddr:=16#C421, Quantity:=1, ComHandle:=ComPort2.handle, TimeOut:=COM2_TIME_OUT, Buffer:=abyBuffer);
	IF RD_HOLD_REGS.Complete THEN
		IF RD_HOLD_REGS.Exception = 0 THEN
			//... и ошибки отсутствуют
			Shnek.MAV:=WORD_FROM_BYTES (ADR (abyBuffer[0]));	// Слово состояния шнека
			Shnek.Qm:=Shnek.MAV * 100.0 / 16383.0;
			tcount:=tcount + 1;
		END_IF
		// Завершаем опрос модуля
		RD_HOLD_REGS (Enable:=FALSE, Buffer:=abyBuffer);	
		Ready:=TRUE;
		xModule:=30;
	END_IF
	
	//======================================================================================
30:	// Постоянное чтение регистра слова состояния STW привода тянущего устройства 
	//======================================================================================
	Ready:=FALSE;
	RD_HOLD_REGS (Enable:=ComPort2.Ready, Mode:=MB_RTU, DevAddr:=ADR_PULLING, FirstAddr:=16#C417, Quantity:=1, ComHandle:=ComPort2.handle, TimeOut:=COM2_TIME_OUT, Buffer:=abyBuffer);
	IF RD_HOLD_REGS.Complete THEN
		// Сбрасываем соединение
		Pulling.Connect:=FALSE;
		IF RD_HOLD_REGS.Exception = 0 THEN
			//... и ошибки отсутствуют
			Pulling.Connect:=TRUE; // Присваиваем
			Pulling.STW:=WORD_FROM_BYTES (ADR (abyBuffer[0]));	// Слово состояния шнека
			
			IF Pulling.STW.3 THEN ALARM_PCHVS.8:=TRUE; END_IF
			IF Pulling.STW.7 THEN ALARM_PCHVS.9:=TRUE; END_IF
			IF Pulling.STW.13 THEN ALARM_PCHVS.10:=TRUE; END_IF
			IF Pulling.STW.14 THEN ALARM_PCHVS.11:=TRUE; END_IF
			IF Pulling.STW.15 THEN ALARM_PCHVS.12:=TRUE; END_IF
			
			tcount:=tcount + 1;
		END_IF
		// Завершаем опрос модуля
		RD_HOLD_REGS (Enable:=FALSE, Buffer:=abyBuffer);	
		Ready:=TRUE;
		xModule:=40;
	END_IF

	//======================================================================================
40:	// Постоянное чтение регистра основного текущего значения MAV тянущего устройства 
	//======================================================================================
	Ready:=FALSE;
	RD_HOLD_REGS (Enable:=ComPort2.Ready, Mode:=MB_RTU, DevAddr:=ADR_PULLING, FirstAddr:=16#C421, Quantity:=1, ComHandle:=ComPort2.handle, TimeOut:=COM2_TIME_OUT, Buffer:=abyBuffer);
	IF RD_HOLD_REGS.Complete THEN
		IF RD_HOLD_REGS.Exception = 0 THEN
			//... и ошибки отсутствуют
			Pulling.MAV:=WORD_FROM_BYTES (ADR (abyBuffer[0]));	// Слово состояния шнека
			Pulling.Speed:=Pulling.MAV *100.0 / 16383.0;
			tcount:=tcount + 1;
		END_IF
		// Завершаем опрос модуля
		RD_HOLD_REGS (Enable:=FALSE, Buffer:=abyBuffer);	
		Ready:=TRUE;
		xModule:=50;					// Продолжение
	END_IF
	
